FUNCTION_BLOCK Explicit_Controller_FCN_BLK
VAR_INPUT
    ssMethodType: SINT;
    MeasuredTankOutputs: ARRAY [0..1] OF LREAL;
    ref: ARRAY [0..1] OF LREAL;
END_VAR

VAR_OUTPUT
    mv: ARRAY [0..1] OF LREAL;
END_VAR

VAR
    last_x_PreviousInput: ARRAY [0..5] OF LREAL;
    last_mv_DSTATE: ARRAY [0..1] OF LREAL;
    Explicit_b_M: ARRAY [0..11] OF LREAL := [0.00012829320734723115,1.0284618689926092E-5,2.4378658054917943E-5,
        9.19840748563352E-5,0.095123941749644919,1.2151957187730602E-6,2.8085799988137366E-5,0.00013352110274451323,
        9.1481345508264347E-5,2.6760937667881709E-5,-1.5083632311296561E-6,0.095123901802077374];
    Explicit_b_Cm: ARRAY [0..11] OF LREAL := [0.15299877600979192,0.0,0.0,0.15299877600979192,0.0,0.0,0.0,0.0,1.0,
        0.0,0.0,1.0];
    Explicit_b_thmin: ARRAY [0..9] OF LREAL := [-10.0,-14.0,-2.608763482112793,-0.757334910684223,-1.0,-1.0,-12.5,
        -17.5,-6.7801207082609904,-11.7277902321632];
    Explicit_b_thmax: ARRAY [0..9] OF LREAL := [20.0,16.0,27.391236517887208,29.242665089315778,1.0,1.0,25.0,20.0,
        17.219879291739009,12.2722097678368];
    b_i1: ARRAY [0..33] OF INT := [1,23,45,67,87,107,128,148,169,191,211,231,251,271,292,310,332,350,369,391,410,431,
        453,472,492,514,535,554,576,596,616,636,657,676];
    b_i2: ARRAY [0..33] OF INT := [22,44,66,86,106,127,147,168,190,210,230,250,270,291,309,331,349,368,390,409,430,
        452,471,491,513,534,553,575,595,615,635,656,675,697];
    Explicit_c_K: ARRAY [0..696] OF LREAL := [2.0611413896907527,1.9955837259660221,0.261375942086798,
        0.36517295006730383,0.154055652781239,0.21525342211788329,20.0,16.0,27.391236517887208,29.242665089315778,
        1.0,1.0,17.219879291739009,12.2722097678368,10.0,14.0,2.608763482112793,0.757334910684223,1.0,1.0,
        6.7801207082609904,11.7277902321632,-2.0611413896907527,10.306132877927066,2.0017312431194147,
        0.3588547626396722,0.208800889557635,20.0,16.0,27.391236517887208,29.242665089315778,1.0,1.0,25.0,
        17.219879291739009,12.2722097678368,10.0,14.0,2.608763482112793,0.757334910684223,1.0,1.0,
        6.7801207082609904,11.7277902321632,-1.9955837259660218,9.9754498249952146,2.0671005215985825,
        0.25507587776500751,0.14778957157873562,20.0,16.0,27.391236517887208,29.242665089315778,1.0,1.0,20.0,
        17.219879291739009,12.2722097678368,10.0,14.0,2.608763482112793,0.757334910684223,1.0,1.0,
        6.7801207082609904,11.7277902321632,-0.2613759420867981,1.9948353088253725,0.36568008759024018,
        0.010244209084743196,0.21578799487811626,20.0,16.0,27.391236517887208,29.242665089315778,1.0,1.0,
        12.2722097678368,10.0,14.0,2.608763482112793,0.757334910684223,1.0,1.0,6.7801207082609904,11.7277902321632,
        -0.36517295006730388,2.0601920598036507,0.26211153239863794,0.15479976076082763,0.014378493331328977,20.0,
        16.0,27.391236517887208,29.242665089315778,1.0,1.0,17.219879291739009,10.0,14.0,2.608763482112793,
        0.757334910684223,1.0,1.0,6.7801207082609904,11.7277902321632,-0.15405565278123903,1.9948283464872751,
        0.77031009910361337,0.3655913731280393,0.21570378618977479,20.0,16.0,27.391236517887208,29.242665089315778,
        1.0,1.0,17.219879291739009,12.2722097678368,10.0,14.0,2.608763482112793,0.757334910684223,1.0,1.0,12.5,
        11.7277902321632,-0.21525342211788326,2.0601821995500464,0.26201367432910744,1.0760008132237195,
        0.154707893627272,20.0,16.0,27.391236517887208,29.242665089315778,1.0,1.0,17.219879291739009,
        12.2722097678368,10.0,14.0,2.608763482112793,0.757334910684223,1.0,1.0,6.7801207082609904,
        -10.306132877927066,2.0028782849354068,0.35771891427389396,0.20764078266896283,20.0,16.0,27.391236517887208,
        29.242665089315778,1.0,1.0,25.0,17.219879291739009,12.2722097678368,10.0,14.0,2.608763482112793,
        0.757334910684223,1.0,1.0,6.7801207082609904,11.7277902321632,-2.0671005215985825,-2.0017312431194143,
        10.31038937822318,9.979316651871887,20.0,16.0,27.391236517887208,29.242665089315778,1.0,1.0,25.0,20.0,
        17.219879291739009,12.2722097678368,10.0,14.0,2.608763482112793,0.757334910684223,1.0,1.0,
        6.7801207082609904,11.7277902321632,-2.0601920598036503,-0.35885476263967225,10.304338652450928,
        0.0078003539108829258,20.0,16.0,27.391236517887208,29.242665089315778,1.0,1.0,25.0,17.219879291739009,10.0,
        14.0,2.608763482112793,0.757334910684223,1.0,1.0,6.7801207082609904,11.7277902321632,-2.0601821995500464,
        -0.20880088955763496,10.303879948828987,1.0708395480624722,20.0,16.0,27.391236517887208,29.242665089315778,
        1.0,1.0,25.0,17.219879291739009,12.2722097678368,10.0,14.0,2.608763482112793,0.757334910684223,1.0,1.0,
        6.7801207082609904,-9.9754498249952128,2.0680301798015472,0.2541304598084248,0.14685003364909435,20.0,16.0,
        27.391236517887208,29.242665089315778,1.0,1.0,20.0,17.219879291739009,12.2722097678368,10.0,14.0,
        2.608763482112793,0.757334910684223,1.0,1.0,6.7801207082609904,-1.9948353088253725,-0.25507587776500751,
        9.97419631577785,0.0040719490329664855,20.0,16.0,27.391236517887208,29.242665089315778,1.0,1.0,20.0,
        12.2722097678368,10.0,14.0,2.608763482112793,0.757334910684223,1.0,1.0,6.7801207082609904,11.7277902321632,
        -1.9948283464872749,-0.14778957157873562,9.9739050689365616,0.76431342623101861,20.0,16.0,
        27.391236517887208,29.242665089315778,1.0,1.0,20.0,17.219879291739009,12.2722097678368,10.0,14.0,
        2.608763482112793,0.757334910684223,1.0,1.0,12.5,11.7277902321632,-0.26211153239863794,-0.36568008759024018,
        0.010993612348099634,0.014947273027453219,20.0,16.0,27.391236517887208,29.242665089315778,1.0,1.0,10.0,14.0,
        2.608763482112793,0.757334910684223,1.0,1.0,6.7801207082609904,11.7277902321632,-0.77031009910361337,
        -0.010244209084743246,1.9947299388091386,0.36567397657122985,0.21578912879523102,20.0,16.0,
        27.391236517887208,29.242665089315778,1.0,1.0,17.219879291739009,12.2722097678368,10.0,14.0,
        2.608763482112793,0.757334910684223,1.0,1.0,12.5,6.7801207082609904,11.7277902321632,-0.26201367432910749,
        -0.21578799487811628,1.0763493615403084,0.010910348192849671,20.0,16.0,27.391236517887208,
        29.242665089315778,1.0,1.0,12.2722097678368,10.0,14.0,2.608763482112793,0.757334910684223,1.0,1.0,
        6.7801207082609904,-0.36559137312803935,-0.15479976076082763,0.77094478261624777,0.014870549898796829,20.0,
        16.0,27.391236517887208,29.242665089315778,1.0,1.0,17.219879291739009,10.0,14.0,2.608763482112793,
        0.757334910684223,1.0,1.0,12.5,11.7277902321632,-1.0760008132237191,-0.014378493331329066,
        2.0600717378634013,0.26211431296869919,0.15480847558724034,20.0,16.0,27.391236517887208,29.242665089315778,
        1.0,1.0,17.219879291739009,12.2722097678368,10.0,14.0,2.608763482112793,0.757334910684223,1.0,1.0,17.5,
        6.7801207082609904,11.7277902321632,-0.15470789362727197,-0.21570378618977476,0.77082285562521369,
        1.0762511309977898,20.0,16.0,27.391236517887208,29.242665089315778,1.0,1.0,17.219879291739009,
        12.2722097678368,10.0,14.0,2.608763482112793,0.757334910684223,1.0,1.0,12.5,-10.310389378223183,
        -2.0028782849354063,9.9801931781643685,20.0,16.0,27.391236517887208,29.242665089315778,1.0,1.0,25.0,20.0,
        17.219879291739009,12.2722097678368,10.0,14.0,2.608763482112793,0.757334910684223,1.0,1.0,
        6.7801207082609904,11.7277902321632,-10.30433865245093,-0.35771891427389391,-10.303732722383751,
        -1.0699095023920164,20.0,16.0,27.391236517887208,29.242665089315778,1.0,1.0,25.0,17.219879291739009,
        12.2722097678368,10.0,14.0,2.608763482112793,0.757334910684223,1.0,1.0,17.5,6.7801207082609904,
        11.7277902321632,-10.303879948828989,-0.20764078266896283,1.0699095023920167,20.0,16.0,27.391236517887208,
        29.242665089315778,1.0,1.0,25.0,17.219879291739009,12.2722097678368,10.0,14.0,2.608763482112793,
        0.757334910684223,1.0,1.0,6.7801207082609904,-9.9793166518718817,-2.0680301798015472,10.311238407241403,
        20.0,16.0,27.391236517887208,29.242665089315778,1.0,1.0,25.0,20.0,17.219879291739009,12.2722097678368,10.0,
        14.0,2.608763482112793,0.757334910684223,1.0,1.0,6.7801207082609904,-2.0600717378634008,-1.0708395480624708,
        -0.0078003539108829232,10.303732722383758,20.0,16.0,27.391236517887208,29.242665089315778,1.0,1.0,25.0,
        17.219879291739009,12.2722097678368,10.0,14.0,2.608763482112793,0.757334910684223,1.0,1.0,17.5,
        6.7801207082609904,11.7277902321632,-9.9741963157778457,-0.2541304598084248,-9.973787635532247,
        -0.76341041484819772,20.0,16.0,27.391236517887208,29.242665089315778,1.0,1.0,20.0,17.219879291739009,
        12.2722097678368,10.0,14.0,2.608763482112793,0.757334910684223,1.0,1.0,12.5,6.7801207082609904,
        -9.9739050689365616,-0.14685003364909435,0.76341041484819783,20.0,16.0,27.391236517887208,
        29.242665089315778,1.0,1.0,20.0,17.219879291739009,12.2722097678368,10.0,14.0,2.608763482112793,
        0.757334910684223,1.0,1.0,12.5,-1.9947299388091386,-0.76431342623101917,-0.0040719490329664846,
        9.9737876355322488,20.0,16.0,27.391236517887208,29.242665089315778,1.0,1.0,20.0,17.219879291739009,
        12.2722097678368,10.0,14.0,2.608763482112793,0.757334910684223,1.0,1.0,12.5,6.7801207082609904,
        11.7277902321632,-0.77094478261624833,-0.36567397657122985,-0.010993612348099681,0.014958980263312462,20.0,
        16.0,27.391236517887208,29.242665089315778,1.0,1.0,17.219879291739009,10.0,14.0,2.608763482112793,
        0.757334910684223,1.0,1.0,12.5,6.7801207082609904,11.7277902321632,-0.26211431296869925,-1.0763493615403084,
        -0.01494727302745312,0.011010054217011499,20.0,16.0,27.391236517887208,29.242665089315778,1.0,1.0,
        12.2722097678368,10.0,14.0,2.608763482112793,0.757334910684223,1.0,1.0,17.5,6.7801207082609904,
        11.7277902321632,-0.77082285562521369,-0.010910348192849697,-0.215789128795231,1.0763150450241359,20.0,16.0,
        27.391236517887208,29.242665089315778,1.0,1.0,17.219879291739009,12.2722097678368,10.0,14.0,
        2.608763482112793,0.757334910684223,1.0,1.0,12.5,6.7801207082609904,-1.0762511309977894,
        -0.15480847558724031,-0.014870549898796815,0.77091609970584685,20.0,16.0,27.391236517887208,
        29.242665089315778,1.0,1.0,17.219879291739009,12.2722097678368,10.0,14.0,2.608763482112793,
        0.757334910684223,1.0,1.0,12.5,17.5,11.7277902321632,-10.31123840724141,-9.98019317816437,20.0,16.0,
        27.391236517887208,29.242665089315778,1.0,1.0,25.0,20.0,17.219879291739009,12.2722097678368,10.0,14.0,
        2.608763482112793,0.757334910684223,1.0,1.0,6.7801207082609904,-0.77091609970584707,-1.0763150450241361,
        -0.011010054217011499,-0.014958980263312384,20.0,16.0,27.391236517887208,29.242665089315778,1.0,1.0,
        17.219879291739009,12.2722097678368,10.0,14.0,2.608763482112793,0.757334910684223,1.0,1.0,12.5,17.5,
        6.7801207082609904,11.7277902321632];
    Explicit_g_H: ARRAY [0..6969] OF LREAL := [-0.10330544107194929,-0.0014745226031521231,0.10246575755178296,
        0.0015946624161439463,0.10330544107194929,0.0014745226031521231,1.0,0.0,0.0,0.0,0.0,0.0,0.0,0.0,-1.0,-0.0,
        -0.0,-0.0,-0.0,-0.0,-0.0,-0.0,0.10330544107194932,-0.090583151736267742,-0.0017962349061867956,
        0.0019086047501879714,0.0017962349061867956,1.0,0.0,0.0,0.0,0.0,0.0,0.0,0.0,0.0,-1.0,-0.0,-0.0,-0.0,-0.0,
        -0.0,-0.0,-0.0,0.0014745226031521231,-0.0020664403881641815,-0.10329574071922931,0.10245558523686728,
        0.10329574071922931,1.0,0.0,0.0,0.0,0.0,0.0,0.0,0.0,0.0,-1.0,-0.0,-0.0,-0.0,-0.0,-0.0,-0.0,-0.0,
        -0.10246575755178298,-0.0016921077114560436,0.0018070761592905537,0.1036139903469729,0.0016921077114560436,
        1.0,0.0,0.0,0.0,0.0,0.0,0.0,-1.0,-0.0,-0.0,-0.0,-0.0,-0.0,-0.0,-0.0,-0.0015946624161439465,
        -0.10329918232016434,0.10245919014615755,0.10329918232016434,0.0013034270519242509,1.0,0.0,0.0,0.0,0.0,0.0,
        0.0,-1.0,-0.0,-0.0,-0.0,-0.0,-0.0,-0.0,-0.0,-0.10330544107194932,-0.0017962349061867956,
        0.090583151736267742,0.0019086047501879714,0.0017962349061867956,1.0,0.0,0.0,0.0,0.0,0.0,0.0,0.0,-1.0,-0.0,
        -0.0,-0.0,-0.0,-0.0,-0.0,-0.0,-0.0014745226031521231,-0.10329574071922931,0.10245558523686728,
        0.0020664403881641815,0.10329574071922931,1.0,0.0,0.0,0.0,0.0,0.0,0.0,0.0,-1.0,-0.0,-0.0,-0.0,-0.0,-0.0,
        -0.0,0.090583151736267686,-0.0018064099095009775,0.00191855841785106,0.0018064099095009775,1.0,0.0,0.0,0.0,
        0.0,0.0,0.0,0.0,0.0,-1.0,-0.0,-0.0,-0.0,-0.0,-0.0,-0.0,-0.0,0.10329574071922928,0.0017962349061867954,
        -0.090574043803180182,-0.0023185749657277268,1.0,0.0,0.0,0.0,0.0,0.0,0.0,0.0,0.0,0.0,-1.0,-0.0,-0.0,-0.0,
        -0.0,-0.0,-0.0,-0.0,0.10329918232016433,-0.0019086047501879714,-0.090577300277252346,0.0016329685799659197,
        1.0,0.0,0.0,0.0,0.0,0.0,0.0,0.0,-1.0,-0.0,-0.0,-0.0,-0.0,-0.0,-0.0,-0.0,0.10329574071922928,
        -0.0017962349061867954,-0.090574043803180182,0.0023185749657277268,1.0,0.0,0.0,0.0,0.0,0.0,0.0,0.0,0.0,-1.0,
        -0.0,-0.0,-0.0,-0.0,-0.0,-0.0,0.0020664403881641823,-0.10329547444997711,0.1024553070868839,
        0.10329547444997711,1.0,0.0,0.0,0.0,0.0,0.0,0.0,0.0,0.0,-1.0,-0.0,-0.0,-0.0,-0.0,-0.0,-0.0,
        0.0016921077114560436,-0.10245558523686726,-0.0022374573065447505,0.10360521588894454,1.0,0.0,0.0,0.0,0.0,
        0.0,0.0,0.0,-1.0,-0.0,-0.0,-0.0,-0.0,-0.0,-0.0,-0.0,0.0017962349061867956,-0.10329574071922931,
        -0.0023185749657277242,0.090574043803180029,1.0,0.0,0.0,0.0,0.0,0.0,0.0,0.0,0.0,-1.0,-0.0,-0.0,-0.0,-0.0,
        -0.0,-0.0,-0.0,-0.10245919014615754,-0.0018070761592905537,0.10360833927584194,0.0015261960444034593,1.0,
        0.0,0.0,0.0,0.0,0.0,-1.0,-0.0,-0.0,-0.0,-0.0,-0.0,-0.0,-0.0,-0.090583151736267686,-0.1036139903469729,
        -0.0018064099095009775,0.00191855841785106,0.0018064099095009775,1.0,0.0,0.0,0.0,0.0,0.0,0.0,0.0,-1.0,-0.0,
        -0.0,-0.0,-0.0,-0.0,-0.0,-0.0,-0.0,-0.10245558523686728,-0.0016921077114560434,0.0022374573065447496,
        0.10360521588894449,1.0,0.0,0.0,0.0,0.0,0.0,0.0,-1.0,-0.0,-0.0,-0.0,-0.0,-0.0,-0.0,-0.0019086047501879716,
        -0.10329918232016436,0.0905773002772523,0.0016329685799659197,1.0,0.0,0.0,0.0,0.0,0.0,0.0,-1.0,-0.0,-0.0,
        -0.0,-0.0,-0.0,-0.0,-0.0,-0.0020664403881641823,-0.0013034270519242512,-0.10329547444997711,
        0.1024553070868839,0.10329547444997711,1.0,0.0,0.0,0.0,0.0,0.0,0.0,0.0,-1.0,-0.0,-0.0,-0.0,-0.0,-0.0,-0.0,
        -0.0,-0.0,-0.10329574071922928,-0.0017962349061867954,0.090574043803180182,0.0023185749657277268,1.0,0.0,
        0.0,0.0,0.0,0.0,0.0,0.0,-1.0,-0.0,-0.0,-0.0,-0.0,-0.0,-0.0,0.090574043803180043,0.0018064099095009773,
        -0.0023266928925573028,1.0,0.0,0.0,0.0,0.0,0.0,0.0,0.0,0.0,0.0,-1.0,-0.0,-0.0,-0.0,-0.0,-0.0,-0.0,-0.0,
        0.090577300277252346,-0.0019185584178510596,0.090573807363914446,-0.0023266928925573006,1.0,0.0,0.0,0.0,0.0,
        0.0,0.0,0.0,0.0,-1.0,-0.0,-0.0,-0.0,-0.0,-0.0,-0.0,-0.0,-0.0,0.090574043803180043,-0.0018064099095009773,
        0.0023266928925573028,1.0,0.0,0.0,0.0,0.0,0.0,0.0,0.0,0.0,-1.0,-0.0,-0.0,-0.0,-0.0,-0.0,-0.0,
        0.0023185749657277264,0.10329547444997711,-0.09057380736391446,1.0,0.0,0.0,0.0,0.0,0.0,0.0,0.0,0.0,0.0,-1.0,
        -0.0,-0.0,-0.0,-0.0,-0.0,-0.0,0.1032954744499771,-0.0023185749657277247,-0.0016329685799659197,
        -0.0905738073639145,1.0,0.0,0.0,0.0,0.0,0.0,0.0,0.0,0.0,-1.0,-0.0,-0.0,-0.0,-0.0,-0.0,-0.0,-0.0,-0.0,
        0.0022374573065447509,-0.1024553070868839,0.0023266928925573015,-0.090573807363914488,1.0,0.0,0.0,0.0,0.0,
        0.0,0.0,0.0,0.0,-1.0,-0.0,-0.0,-0.0,-0.0,-0.0,-0.0,-0.0,0.0023185749657277255,-0.1032954744499771,
        0.0905738073639145,1.0,0.0,0.0,0.0,0.0,0.0,0.0,0.0,0.0,-1.0,-0.0,-0.0,-0.0,-0.0,-0.0,-0.0,
        0.0018064099095009777,-0.090574043803180057,-0.10360521588894456,-0.0023266928925573011,1.0,0.0,0.0,0.0,0.0,
        0.0,0.0,0.0,0.0,-1.0,-0.0,-0.0,-0.0,-0.0,-0.0,-0.0,-0.0,-0.0,-0.090577300277252318,-0.0019185584178510599,
        -0.10360833927584194,0.0016433588476607495,1.0,0.0,0.0,0.0,0.0,0.0,0.0,-1.0,-0.0,-0.0,-0.0,-0.0,-0.0,-0.0,
        -0.0,-0.0,-0.10245530708688391,-0.0022374573065447492,-0.0015261960444034593,0.10360497454409653,1.0,0.0,
        0.0,0.0,0.0,0.0,0.0,-1.0,-0.0,-0.0,-0.0,-0.0,-0.0,-0.0,-0.0,-0.0,-0.090574043803180043,-0.10360521588894456,
        -0.0018064099095009773,0.0023266928925573028,1.0,0.0,0.0,0.0,0.0,0.0,0.0,0.0,-1.0,-0.0,-0.0,-0.0,-0.0,-0.0,
        -0.0,-0.0,-0.0023185749657277264,-0.10329547444997711,-0.0016329685799659191,0.09057380736391446,1.0,0.0,
        0.0,0.0,0.0,0.0,0.0,0.0,-1.0,-0.0,-0.0,-0.0,-0.0,-0.0,-0.0,-0.0,-0.0,0.090573807363914446,
        0.0023266928925572993,1.0,0.0,0.0,0.0,0.0,0.0,0.0,0.0,0.0,0.0,-1.0,-0.0,-0.0,-0.0,-0.0,-0.0,-0.0,
        -0.090573807363914446,-0.0023266928925572993,-0.10360497454409655,-0.0016433588476607497,1.0,0.0,0.0,0.0,
        0.0,0.0,0.0,0.0,-1.0,-0.0,-0.0,-0.0,-0.0,-0.0,-0.0,-0.0,-0.0,-0.0,-0.0029866651271786876,
        -0.10390116291611282,0.0031875003616156274,0.10304688647343455,0.0029866651271786876,0.10390116291611282,
        0.0,1.0,0.0,0.0,0.0,0.0,0.0,0.0,-0.0,-1.0,-0.0,-0.0,-0.0,-0.0,-0.0,-0.0,0.002986665127178688,
        -0.0039359133245656739,-0.10389613523146926,0.1030418390266099,0.10389613523146926,0.0,1.0,0.0,0.0,0.0,0.0,
        0.0,0.0,0.0,-0.0,-1.0,-0.0,-0.0,-0.0,-0.0,-0.0,-0.0,0.10390116291611282,-0.091095658056062873,
        -0.0033113868084985666,0.0035130907390366621,0.0033113868084985666,0.0,1.0,0.0,0.0,0.0,0.0,0.0,0.0,0.0,-0.0,
        -1.0,-0.0,-0.0,-0.0,-0.0,-0.0,-0.0,-0.0031875003616156279,-0.1038978860866369,0.10304359668322663,
        0.0026964566969657241,0.1038978860866369,0.0,1.0,0.0,0.0,0.0,0.0,0.0,-0.0,-1.0,-0.0,-0.0,-0.0,-0.0,-0.0,
        -0.0,-0.10304688647343456,-0.0032003930853852416,0.0034018852466296103,0.0032003930853852416,
        0.10422852726420227,0.0,1.0,0.0,0.0,0.0,0.0,0.0,-0.0,-1.0,-0.0,-0.0,-0.0,-0.0,-0.0,-0.0,
        -0.002986665127178688,-0.10389613523146926,0.0039359133245656739,0.1030418390266099,0.10389613523146926,0.0,
        1.0,0.0,0.0,0.0,0.0,0.0,0.0,-0.0,-1.0,-0.0,-0.0,-0.0,-0.0,-0.0,-0.0,-0.10390116291611282,
        -0.0033113868084985666,0.0035130907390366621,0.091095658056062873,0.0033113868084985666,0.0,1.0,0.0,0.0,0.0,
        0.0,0.0,0.0,-0.0,-1.0,-0.0,-0.0,-0.0,-0.0,-0.0,0.0039359133245656722,-0.10389596374005793,
        0.10304166986211653,0.10389596374005793,0.0,1.0,0.0,0.0,0.0,0.0,0.0,0.0,0.0,-0.0,-1.0,-0.0,-0.0,-0.0,-0.0,
        -0.0,-0.0,0.0033113868084985666,0.10389613523146926,-0.0042412342413153167,-0.091092939463560868,0.0,1.0,
        0.0,0.0,0.0,0.0,0.0,0.0,0.0,0.0,-0.0,-1.0,-0.0,-0.0,-0.0,-0.0,-0.0,-0.0,0.0032003930853852407,
        -0.10304183902660989,-0.0041373691182175487,0.10422380845249599,0.0,1.0,0.0,0.0,0.0,0.0,0.0,0.0,-0.0,-1.0,
        -0.0,-0.0,-0.0,-0.0,-0.0,-0.0,0.0033113868084985666,-0.10389613523146926,-0.0042412342413153167,
        0.091092939463560868,0.0,1.0,0.0,0.0,0.0,0.0,0.0,0.0,0.0,-0.0,-1.0,-0.0,-0.0,-0.0,-0.0,-0.0,
        0.091095658056062873,-0.0033199458639416968,0.0035216972663637824,0.0033199458639416968,0.0,1.0,0.0,0.0,0.0,
        0.0,0.0,0.0,0.0,-0.0,-1.0,-0.0,-0.0,-0.0,-0.0,-0.0,0.10389788608663691,-0.0035130907390366617,
        -0.0910939728911974,0.0030174925306511403,0.0,1.0,0.0,0.0,0.0,0.0,0.0,0.0,-0.0,-1.0,-0.0,-0.0,-0.0,-0.0,
        -0.0,-0.0,0.10389613523146925,-0.0033113868084985666,-0.091092939463560924,0.0042412342413153123,0.0,1.0,
        0.0,0.0,0.0,0.0,0.0,0.0,0.0,-0.0,-1.0,-0.0,-0.0,-0.0,-0.0,-0.0,-0.0,-0.0034018852466296103,
        -0.10304359668322662,0.0029076453649676762,0.10422546298600668,0.0,1.0,0.0,0.0,0.0,0.0,-0.0,-1.0,-0.0,-0.0,
        -0.0,-0.0,-0.0,-0.0,-0.0039359133245656722,-0.0026964566969657237,-0.10389596374005793,0.10304166986211653,
        0.10389596374005793,0.0,1.0,0.0,0.0,0.0,0.0,0.0,0.0,-0.0,-1.0,-0.0,-0.0,-0.0,-0.0,-0.0,-0.0,-0.0,
        -0.0035130907390366621,-0.1038978860866369,0.091093972891197583,0.0030174925306511377,0.0,1.0,0.0,0.0,0.0,
        0.0,0.0,-0.0,-1.0,-0.0,-0.0,-0.0,-0.0,-0.0,-0.1030418390266099,-0.0032003930853852416,0.0041373691182175461,
        0.10422380845249597,0.0,1.0,0.0,0.0,0.0,0.0,0.0,-0.0,-1.0,-0.0,-0.0,-0.0,-0.0,-0.0,-0.0,
        -0.091095658056062873,-0.10422852726420226,-0.0033199458639416968,0.0035216972663637824,
        0.0033199458639416968,0.0,1.0,0.0,0.0,0.0,0.0,0.0,0.0,-0.0,-1.0,-0.0,-0.0,-0.0,-0.0,-0.0,-0.0,-0.0,
        -0.0033113868084985666,-0.10389613523146926,0.0042412342413153167,0.091092939463560868,0.0,1.0,0.0,0.0,0.0,
        0.0,0.0,0.0,-0.0,-1.0,-0.0,-0.0,-0.0,-0.0,-0.0,0.0042412342413153149,0.10389596374005791,
        -0.09109287411848567,0.0,1.0,0.0,0.0,0.0,0.0,0.0,0.0,0.0,0.0,-0.0,-1.0,-0.0,-0.0,-0.0,-0.0,-0.0,-0.0,
        0.0041373691182175452,-0.10304166986211651,0.0042494263649640318,-0.0910928741184855,0.0,1.0,0.0,0.0,0.0,
        0.0,0.0,0.0,0.0,-0.0,-1.0,-0.0,-0.0,-0.0,-0.0,-0.0,-0.0,-0.0,0.0042412342413153149,-0.10389596374005791,
        0.09109287411848567,0.0,1.0,0.0,0.0,0.0,0.0,0.0,0.0,0.0,-0.0,-1.0,-0.0,-0.0,-0.0,-0.0,-0.0,
        0.0910929394635609,0.0033199458639416963,-0.0042494263649640335,0.0,1.0,0.0,0.0,0.0,0.0,0.0,0.0,0.0,0.0,
        -0.0,-1.0,-0.0,-0.0,-0.0,-0.0,-0.0,0.0033199458639416959,-0.091092939463561,-0.10422380845249592,
        -0.004249426364964037,0.0,1.0,0.0,0.0,0.0,0.0,0.0,0.0,0.0,-0.0,-1.0,-0.0,-0.0,-0.0,-0.0,-0.0,-0.0,-0.0,
        0.0910939728911976,-0.0035216972663637829,0.091092874118485587,-0.0042494263649640309,0.0,1.0,0.0,0.0,0.0,
        0.0,0.0,0.0,0.0,-0.0,-1.0,-0.0,-0.0,-0.0,-0.0,-0.0,-0.0,0.0910929394635609,-0.0033199458639416968,
        0.0042494263649640318,0.0,1.0,0.0,0.0,0.0,0.0,0.0,0.0,0.0,-0.0,-1.0,-0.0,-0.0,-0.0,-0.0,-0.0,
        0.10389596374005794,-0.0042412342413153132,-0.0030174925306511394,-0.091092874118485587,0.0,1.0,0.0,0.0,0.0,
        0.0,0.0,0.0,0.0,-0.0,-1.0,-0.0,-0.0,-0.0,-0.0,-0.0,-0.0,-0.0,-0.0041373691182175444,-0.10304166986211653,
        -0.0029076453649676775,0.10422364519688854,0.0,1.0,0.0,0.0,0.0,0.0,0.0,-0.0,-1.0,-0.0,-0.0,-0.0,-0.0,-0.0,
        -0.0,-0.0,-0.0035216972663637833,-0.091093972891197486,-0.10422546298600667,0.00302592181600906,0.0,1.0,0.0,
        0.0,0.0,0.0,0.0,-0.0,-1.0,-0.0,-0.0,-0.0,-0.0,-0.0,-0.0,-0.0,-0.0042412342413153149,-0.0030174925306511386,
        -0.10389596374005791,0.09109287411848567,0.0,1.0,0.0,0.0,0.0,0.0,0.0,0.0,-0.0,-1.0,-0.0,-0.0,-0.0,-0.0,-0.0,
        -0.0,-0.0910929394635609,-0.0033199458639416963,-0.10422380845249594,0.0042494263649640335,0.0,1.0,0.0,0.0,
        0.0,0.0,0.0,0.0,-0.0,-1.0,-0.0,-0.0,-0.0,-0.0,-0.0,-0.0,-0.0,0.0042494263649640335,0.091092874118485545,0.0,
        1.0,0.0,0.0,0.0,0.0,0.0,0.0,0.0,0.0,-0.0,-1.0,-0.0,-0.0,-0.0,-0.0,-0.0,-0.0042494263649640335,
        -0.091092874118485545,-0.00302592181600906,-0.10422364519688854,0.0,1.0,0.0,0.0,0.0,0.0,0.0,0.0,-0.0,-1.0,
        -0.0,-0.0,-0.0,-0.0,-0.0,-0.0,-0.0,-0.0,-0.0071014157036083953,-0.00011441872526747157,
        0.0068071732563204012,0.00012053113664926074,0.0071014157036083953,0.00011441872526747157,0.0,0.0,1.0,0.0,
        0.0,0.0,0.0,0.0,-0.0,-0.0,-1.0,-0.0,-0.0,-0.0,-0.0,-0.0,0.0071014157036083962,-0.0048430438770123655,
        -0.00013653204941286985,0.00014211064337640565,0.00013653204941286985,0.0,0.0,1.0,0.0,0.0,0.0,0.0,0.0,0.0,
        -0.0,-0.0,-1.0,-0.0,-0.0,-0.0,-0.0,-0.0,0.00011441872526747157,-0.000141573042344912,-0.0071007897421819293,
        0.0068065491278817619,0.0071007897421819293,0.0,0.0,1.0,0.0,0.0,0.0,0.0,0.0,0.0,-0.0,-0.0,-1.0,-0.0,-0.0,
        -0.0,-0.0,-0.0,-0.0068071732563204021,-0.00012887210385476621,0.00013464115259381751,0.0074369160608808611,
        0.00012887210385476621,0.0,0.0,1.0,0.0,0.0,0.0,0.0,-0.0,-0.0,-1.0,-0.0,-0.0,-0.0,-0.0,-0.0,
        -0.00012053113664926074,-0.0071010081244634151,0.00680676736109825,0.0071010081244634151,
        0.00010540752661209963,0.0,0.0,1.0,0.0,0.0,0.0,0.0,-0.0,-0.0,-1.0,-0.0,-0.0,-0.0,-0.0,-0.0,
        -0.0071014157036083962,-0.00013653204941286985,0.0048430438770123655,0.00014211064337640565,
        0.00013653204941286985,0.0,0.0,1.0,0.0,0.0,0.0,0.0,0.0,-0.0,-0.0,-1.0,-0.0,-0.0,-0.0,-0.0,-0.0,
        -0.00011441872526747157,-0.0071007897421819293,0.0068065491278817619,0.000141573042344912,
        0.0071007897421819293,0.0,0.0,1.0,0.0,0.0,0.0,0.0,0.0,-0.0,-0.0,-1.0,-0.0,-0.0,-0.0,-0.0,
        0.004843043877012362,-0.0001370758183784174,0.00014264258380223117,0.0001370758183784174,0.0,0.0,1.0,0.0,
        0.0,0.0,0.0,0.0,0.0,-0.0,-0.0,-1.0,-0.0,-0.0,-0.0,-0.0,-0.0,0.0071007897421819293,0.00013653204941286982,
        -0.00484267616986334,-0.00015890541712753912,0.0,0.0,1.0,0.0,0.0,0.0,0.0,0.0,0.0,0.0,-0.0,-0.0,-1.0,-0.0,
        -0.0,-0.0,-0.0,-0.0,0.0071010081244634142,-0.00014211064337640562,-0.0048428095237973432,
        0.00012805865559832721,0.0,0.0,1.0,0.0,0.0,0.0,0.0,0.0,-0.0,-0.0,-1.0,-0.0,-0.0,-0.0,-0.0,-0.0,
        0.0071007897421819293,-0.00013653204941286982,-0.00484267616986334,0.00015890541712753912,0.0,0.0,1.0,0.0,
        0.0,0.0,0.0,0.0,0.0,-0.0,-0.0,-1.0,-0.0,-0.0,-0.0,-0.0,0.00014157304234491195,-0.0071007713931416907,
        0.0068065310553807263,0.0071007713931416907,0.0,0.0,1.0,0.0,0.0,0.0,0.0,0.0,0.0,-0.0,-0.0,-1.0,-0.0,-0.0,
        -0.0,-0.0,0.00012887210385476621,-0.006806549127881761,-0.00015293404910673837,0.0074363092277326959,0.0,
        0.0,1.0,0.0,0.0,0.0,0.0,0.0,-0.0,-0.0,-1.0,-0.0,-0.0,-0.0,-0.0,-0.0,0.00013653204941286982,
        -0.00710078974218193,-0.00015890541712753893,0.0048426761698633393,0.0,0.0,1.0,0.0,0.0,0.0,0.0,0.0,0.0,-0.0,
        -0.0,-1.0,-0.0,-0.0,-0.0,-0.0,-0.0,-0.0068067673610982512,-0.00013464115259381751,0.0074365205859498427,
        0.0001202050585799296,0.0,0.0,1.0,0.0,0.0,0.0,-0.0,-0.0,-1.0,-0.0,-0.0,-0.0,-0.0,-0.0,-0.004843043877012362,
        -0.0074369160608808611,-0.0001370758183784174,0.00014264258380223117,0.0001370758183784174,0.0,0.0,1.0,0.0,
        0.0,0.0,0.0,0.0,-0.0,-0.0,-1.0,-0.0,-0.0,-0.0,-0.0,-0.0,-0.0,-0.0068065491278817619,-0.00012887210385476621,
        0.00015293404910673842,0.0074363092277326941,0.0,0.0,1.0,0.0,0.0,0.0,0.0,-0.0,-0.0,-1.0,-0.0,-0.0,-0.0,-0.0,
        -0.00014211064337640565,-0.0071010081244634159,0.0048428095237973406,0.00012805865559832721,0.0,0.0,1.0,0.0,
        0.0,0.0,0.0,-0.0,-0.0,-1.0,-0.0,-0.0,-0.0,-0.0,-0.0,-0.00014157304234491195,-0.00010540752661209965,
        -0.0071007713931416907,0.0068065310553807263,0.0071007713931416907,0.0,0.0,1.0,0.0,0.0,0.0,0.0,0.0,-0.0,
        -0.0,-1.0,-0.0,-0.0,-0.0,-0.0,-0.0,-0.0,-0.0071007897421819293,-0.00013653204941286982,0.00484267616986334,
        0.00015890541712753912,0.0,0.0,1.0,0.0,0.0,0.0,0.0,0.0,-0.0,-0.0,-1.0,-0.0,-0.0,-0.0,-0.0,
        0.0048426761698633488,0.0001370758183784174,-0.00015933928310827815,0.0,0.0,1.0,0.0,0.0,0.0,0.0,0.0,0.0,0.0,
        -0.0,-0.0,-1.0,-0.0,-0.0,-0.0,-0.0,-0.0,0.0048428095237973475,-0.00014264258380223112,0.0048426666784349339,
        -0.00015933928310827783,0.0,0.0,1.0,0.0,0.0,0.0,0.0,0.0,0.0,-0.0,-0.0,-1.0,-0.0,-0.0,-0.0,-0.0,-0.0,-0.0,
        0.0048426761698633488,-0.0001370758183784174,0.00015933928310827815,0.0,0.0,1.0,0.0,0.0,0.0,0.0,0.0,0.0,
        -0.0,-0.0,-1.0,-0.0,-0.0,-0.0,-0.0,0.00015890541712753904,0.0071007713931416925,-0.0048426666784349322,0.0,
        0.0,1.0,0.0,0.0,0.0,0.0,0.0,0.0,0.0,-0.0,-0.0,-1.0,-0.0,-0.0,-0.0,-0.0,0.00710077139314169,
        -0.00015890541712753904,-0.00012805865559832719,-0.0048426666784349417,0.0,0.0,1.0,0.0,0.0,0.0,0.0,0.0,0.0,
        -0.0,-0.0,-1.0,-0.0,-0.0,-0.0,-0.0,-0.0,-0.0,0.00015293404910673837,-0.0068065310553807254,
        0.000159339283108278,-0.0048426666784349304,0.0,0.0,1.0,0.0,0.0,0.0,0.0,0.0,0.0,-0.0,-0.0,-1.0,-0.0,-0.0,
        -0.0,-0.0,-0.0,0.000158905417127539,-0.00710077139314169,0.0048426666784349348,0.0,0.0,1.0,0.0,0.0,0.0,0.0,
        0.0,0.0,-0.0,-0.0,-1.0,-0.0,-0.0,-0.0,-0.0,0.0001370758183784174,-0.0048426761698633454,
        -0.0074363092277326967,-0.0001593392831082781,0.0,0.0,1.0,0.0,0.0,0.0,0.0,0.0,0.0,-0.0,-0.0,-1.0,-0.0,-0.0,
        -0.0,-0.0,-0.0,-0.0,-0.0048428095237973458,-0.00014264258380223115,-0.0074365205859498436,
        0.00012861393248801036,0.0,0.0,1.0,0.0,0.0,0.0,0.0,-0.0,-0.0,-1.0,-0.0,-0.0,-0.0,-0.0,-0.0,-0.0,
        -0.0068065310553807271,-0.00015293404910673839,-0.00012020505857992958,0.0074362911951540191,0.0,0.0,1.0,
        0.0,0.0,0.0,0.0,-0.0,-0.0,-1.0,-0.0,-0.0,-0.0,-0.0,-0.0,-0.0,-0.0048426761698633488,-0.007436309227732695,
        -0.0001370758183784174,0.00015933928310827815,0.0,0.0,1.0,0.0,0.0,0.0,0.0,0.0,-0.0,-0.0,-1.0,-0.0,-0.0,-0.0,
        -0.0,-0.0,-0.00015890541712753904,-0.0071007713931416925,-0.00012805865559832716,0.0048426666784349322,0.0,
        0.0,1.0,0.0,0.0,0.0,0.0,0.0,-0.0,-0.0,-1.0,-0.0,-0.0,-0.0,-0.0,-0.0,-0.0,0.004842666678434933,
        0.00015933928310827788,0.0,0.0,1.0,0.0,0.0,0.0,0.0,0.0,0.0,0.0,-0.0,-0.0,-1.0,-0.0,-0.0,-0.0,-0.0,
        -0.004842666678434933,-0.00015933928310827788,-0.00743629119515402,-0.00012861393248801042,0.0,0.0,1.0,0.0,
        0.0,0.0,0.0,0.0,-0.0,-0.0,-1.0,-0.0,-0.0,-0.0,-0.0,-0.0,-0.0,-0.0,-0.00040913205147735833,
        -0.012803913199114694,0.00042684709847512454,0.012280530787446623,0.00040913205147735833,
        0.012803913199114694,0.0,0.0,0.0,1.0,0.0,0.0,0.0,0.0,-0.0,-0.0,-0.0,-1.0,-0.0,-0.0,-0.0,-0.0,
        0.00040913205147735839,-0.00048184876971232865,-0.012803421641857477,0.012280091043666855,
        0.012803421641857477,0.0,0.0,0.0,1.0,0.0,0.0,0.0,0.0,0.0,-0.0,-0.0,-0.0,-1.0,-0.0,-0.0,-0.0,-0.0,
        0.012803913199114692,-0.0087802267724355568,-0.00044914235230113112,0.00046696522506884096,
        0.00044914235230113112,0.0,0.0,0.0,1.0,0.0,0.0,0.0,0.0,0.0,-0.0,-0.0,-0.0,-1.0,-0.0,-0.0,-0.0,-0.0,
        -0.00042684709847512465,-0.012803581733992975,0.012280236188633492,0.00038239527547962392,
        0.012803581733992975,0.0,0.0,0.0,1.0,0.0,0.0,0.0,-0.0,-0.0,-0.0,-1.0,-0.0,-0.0,-0.0,-0.0,
        -0.012280530787446625,-0.00043459798254794492,0.00045239171239116143,0.00043459798254794492,
        0.013399805276596607,0.0,0.0,0.0,1.0,0.0,0.0,0.0,-0.0,-0.0,-0.0,-1.0,-0.0,-0.0,-0.0,-0.0,
        -0.00040913205147735839,-0.012803421641857477,0.00048184876971232865,0.012280091043666855,
        0.012803421641857477,0.0,0.0,0.0,1.0,0.0,0.0,0.0,0.0,-0.0,-0.0,-0.0,-1.0,-0.0,-0.0,-0.0,-0.0,
        -0.012803913199114692,-0.00044914235230113112,0.00046696522506884096,0.0087802267724355568,
        0.00044914235230113112,0.0,0.0,0.0,1.0,0.0,0.0,0.0,0.0,-0.0,-0.0,-0.0,-1.0,-0.0,-0.0,-0.0,
        0.00048184876971232816,-0.012803400150311305,0.012280072289609674,0.012803400150311305,0.0,0.0,0.0,1.0,0.0,
        0.0,0.0,0.0,0.0,-0.0,-0.0,-0.0,-1.0,-0.0,-0.0,-0.0,-0.0,0.00044914235230113112,0.012803421641857476,
        -0.00051947485679715278,-0.0087802823071337216,0.0,0.0,0.0,1.0,0.0,0.0,0.0,0.0,0.0,0.0,-0.0,-0.0,-0.0,-1.0,
        -0.0,-0.0,-0.0,-0.0,0.00043459798254794486,-0.012280091043666853,-0.00050585606663743662,
        0.013399272511122719,0.0,0.0,0.0,1.0,0.0,0.0,0.0,0.0,-0.0,-0.0,-0.0,-1.0,-0.0,-0.0,-0.0,-0.0,
        0.00044914235230113112,-0.012803421641857476,-0.00051947485679715278,0.0087802823071337216,0.0,0.0,0.0,1.0,
        0.0,0.0,0.0,0.0,0.0,-0.0,-0.0,-0.0,-1.0,-0.0,-0.0,-0.0,0.00878022677243555,-0.00044996673444029655,
        0.000467794169019148,0.00044996673444029655,0.0,0.0,0.0,1.0,0.0,0.0,0.0,0.0,0.0,-0.0,-0.0,-0.0,-1.0,-0.0,
        -0.0,-0.0,0.012803581733992975,-0.00046696522506884091,-0.0087802788142219718,0.00042195050475040259,0.0,
        0.0,0.0,1.0,0.0,0.0,0.0,0.0,-0.0,-0.0,-0.0,-1.0,-0.0,-0.0,-0.0,-0.0,0.012803421641857476,
        -0.00044914235230113117,-0.0087802823071337164,0.00051947485679715191,0.0,0.0,0.0,1.0,0.0,0.0,0.0,0.0,0.0,
        -0.0,-0.0,-0.0,-1.0,-0.0,-0.0,-0.0,-0.0,-0.00045239171239116148,-0.012280236188633491,
        0.00040755820299425842,0.013399444045468174,0.0,0.0,0.0,1.0,0.0,0.0,-0.0,-0.0,-0.0,-1.0,-0.0,-0.0,-0.0,-0.0,
        -0.00048184876971232816,-0.000382395275479624,-0.012803400150311305,0.012280072289609674,
        0.012803400150311305,0.0,0.0,0.0,1.0,0.0,0.0,0.0,0.0,-0.0,-0.0,-0.0,-1.0,-0.0,-0.0,-0.0,-0.0,-0.0,
        -0.00046696522506884091,-0.012803581733992975,0.0087802788142219822,0.00042195050475040254,0.0,0.0,0.0,1.0,
        0.0,0.0,0.0,-0.0,-0.0,-0.0,-1.0,-0.0,-0.0,-0.0,-0.012280091043666855,-0.00043459798254794492,
        0.00050585606663743629,0.013399272511122717,0.0,0.0,0.0,1.0,0.0,0.0,0.0,-0.0,-0.0,-0.0,-1.0,-0.0,-0.0,-0.0,
        -0.0,-0.00878022677243555,-0.013399805276596607,-0.00044996673444029655,0.000467794169019148,
        0.00044996673444029655,0.0,0.0,0.0,1.0,0.0,0.0,0.0,0.0,-0.0,-0.0,-0.0,-1.0,-0.0,-0.0,-0.0,-0.0,-0.0,
        -0.00044914235230113112,-0.012803421641857476,0.00051947485679715278,0.0087802823071337216,0.0,0.0,0.0,1.0,
        0.0,0.0,0.0,0.0,-0.0,-0.0,-0.0,-1.0,-0.0,-0.0,-0.0,0.00051947485679715256,0.012803400150311308,
        -0.0087802859415915882,0.0,0.0,0.0,1.0,0.0,0.0,0.0,0.0,0.0,0.0,-0.0,-0.0,-0.0,-1.0,-0.0,-0.0,-0.0,-0.0,
        0.00050585606663743619,-0.012280072289609669,0.00052026393633152477,-0.00878028594159158,0.0,0.0,0.0,1.0,
        0.0,0.0,0.0,0.0,0.0,-0.0,-0.0,-0.0,-1.0,-0.0,-0.0,-0.0,-0.0,-0.0,0.00051947485679715256,
        -0.012803400150311308,0.0087802859415915882,0.0,0.0,0.0,1.0,0.0,0.0,0.0,0.0,0.0,-0.0,-0.0,-0.0,-1.0,-0.0,
        -0.0,-0.0,0.0087802823071337164,0.00044996673444029644,-0.0005202639363315252,0.0,0.0,0.0,1.0,0.0,0.0,0.0,
        0.0,0.0,0.0,-0.0,-0.0,-0.0,-1.0,-0.0,-0.0,-0.0,0.00044996673444029655,-0.0087802823071337112,
        -0.013399272511122719,-0.00052026393633152455,0.0,0.0,0.0,1.0,0.0,0.0,0.0,0.0,0.0,-0.0,-0.0,-0.0,-1.0,-0.0,
        -0.0,-0.0,-0.0,-0.0,0.0087802788142219909,-0.00046779416901914796,0.0087802859415916073,
        -0.00052026393633152531,0.0,0.0,0.0,1.0,0.0,0.0,0.0,0.0,0.0,-0.0,-0.0,-0.0,-1.0,-0.0,-0.0,-0.0,-0.0,
        0.0087802823071337233,-0.0004499667344402965,0.00052026393633152542,0.0,0.0,0.0,1.0,0.0,0.0,0.0,0.0,0.0,
        -0.0,-0.0,-0.0,-1.0,-0.0,-0.0,-0.0,0.012803400150311306,-0.00051947485679715234,-0.0004219505047504027,
        -0.0087802859415915917,0.0,0.0,0.0,1.0,0.0,0.0,0.0,0.0,0.0,-0.0,-0.0,-0.0,-1.0,-0.0,-0.0,-0.0,-0.0,-0.0,
        -0.000505856066637436,-0.012280072289609674,-0.00040755820299425859,0.013399248530954264,0.0,0.0,0.0,1.0,
        0.0,0.0,0.0,-0.0,-0.0,-0.0,-1.0,-0.0,-0.0,-0.0,-0.0,-0.0,-0.000467794169019148,-0.0087802788142219753,
        -0.013399444045468176,0.00042276241085400672,0.0,0.0,0.0,1.0,0.0,0.0,0.0,-0.0,-0.0,-0.0,-1.0,-0.0,-0.0,-0.0,
        -0.0,-0.0,-0.00051947485679715256,-0.00042195050475040254,-0.012803400150311308,0.0087802859415915882,0.0,
        0.0,0.0,1.0,0.0,0.0,0.0,0.0,-0.0,-0.0,-0.0,-1.0,-0.0,-0.0,-0.0,-0.0,-0.0087802823071337164,
        -0.00044996673444029644,-0.013399272511122716,0.0005202639363315252,0.0,0.0,0.0,1.0,0.0,0.0,0.0,0.0,-0.0,
        -0.0,-0.0,-1.0,-0.0,-0.0,-0.0,-0.0,-0.0,0.00052026393633152488,0.0087802859415915847,0.0,0.0,0.0,1.0,0.0,
        0.0,0.0,0.0,0.0,0.0,-0.0,-0.0,-0.0,-1.0,-0.0,-0.0,-0.0,-0.00052026393633152488,-0.0087802859415915847,
        -0.00042276241085400677,-0.013399248530954271,0.0,0.0,0.0,1.0,0.0,0.0,0.0,0.0,-0.0,-0.0,-0.0,-1.0,-0.0,-0.0,
        -0.0,-0.0,-0.0,-0.0,-0.699842938730663,-0.010035599503395155,0.69332035945645,0.010841852728168152,
        0.699842938730663,0.010035599503395155,0.0,0.0,0.0,0.0,1.0,0.0,0.0,0.0,-0.0,-0.0,-0.0,-0.0,-1.0,-0.0,-0.0,
        -0.0,0.69984293873066306,-0.60877543705459958,-0.012215033803492436,0.012968650442024339,
        0.012215033803492436,0.0,0.0,0.0,0.0,1.0,0.0,0.0,0.0,0.0,-0.0,-0.0,-0.0,-0.0,-1.0,-0.0,-0.0,-0.0,
        0.010035599503395155,-0.013997402719325952,-0.69977736900234788,0.6932517133063042,0.69977736900234788,0.0,
        0.0,0.0,0.0,1.0,0.0,0.0,0.0,0.0,-0.0,-0.0,-0.0,-0.0,-1.0,-0.0,-0.0,-0.0,-0.6933203594564501,
        -0.01150785335521526,0.0122791159302254,0.703041617134732,0.01150785335521526,0.0,0.0,0.0,0.0,1.0,0.0,0.0,
        -0.0,-0.0,-0.0,-0.0,-1.0,-0.0,-0.0,-0.0,-0.010841852728168152,-0.69980061939953575,0.69327602991798487,
        0.69980061939953575,0.0088862950073843542,0.0,0.0,0.0,0.0,1.0,0.0,0.0,-0.0,-0.0,-0.0,-0.0,-1.0,-0.0,-0.0,
        -0.0,-0.69984293873066306,-0.012215033803492436,0.60877543705459958,0.012968650442024339,
        0.012215033803492436,0.0,0.0,0.0,0.0,1.0,0.0,0.0,0.0,-0.0,-0.0,-0.0,-0.0,-1.0,-0.0,-0.0,-0.0,
        -0.010035599503395155,-0.69977736900234788,0.6932517133063042,0.013997402719325952,0.69977736900234788,0.0,
        0.0,0.0,0.0,1.0,0.0,0.0,0.0,-0.0,-0.0,-0.0,-0.0,-1.0,-0.0,-0.0,0.60877543705459958,-0.012283415343526595,
        0.0130355444868211,0.012283415343526595,0.0,0.0,0.0,0.0,1.0,0.0,0.0,0.0,0.0,-0.0,-0.0,-0.0,-0.0,-1.0,-0.0,
        -0.0,-0.0,0.69977736900234788,0.012215033803492436,-0.60871464776796336,-0.015705489529037081,0.0,0.0,0.0,
        0.0,1.0,0.0,0.0,0.0,0.0,0.0,-0.0,-0.0,-0.0,-0.0,-1.0,-0.0,-0.0,-0.0,0.69980061939953575,
        -0.012968650442024337,-0.60873638906724648,0.011118767018001796,0.0,0.0,0.0,0.0,1.0,0.0,0.0,0.0,-0.0,-0.0,
        -0.0,-0.0,-1.0,-0.0,-0.0,-0.0,0.69977736900234788,-0.012215033803492436,-0.60871464776796336,
        0.015705489529037081,0.0,0.0,0.0,0.0,1.0,0.0,0.0,0.0,0.0,-0.0,-0.0,-0.0,-0.0,-1.0,-0.0,-0.0,
        0.013997402719325936,-0.699775564999848,0.69324983267331119,0.699775564999848,0.0,0.0,0.0,0.0,1.0,0.0,0.0,
        0.0,0.0,-0.0,-0.0,-0.0,-0.0,-1.0,-0.0,-0.0,0.011507853355215258,-0.69325171330630408,-0.015154564068334616,
        0.70298216286030424,0.0,0.0,0.0,0.0,1.0,0.0,0.0,0.0,-0.0,-0.0,-0.0,-0.0,-1.0,-0.0,-0.0,-0.0,
        0.012215033803492434,-0.69977736900234788,-0.015705489529037078,0.60871464776796369,0.0,0.0,0.0,0.0,1.0,0.0,
        0.0,0.0,0.0,-0.0,-0.0,-0.0,-0.0,-1.0,-0.0,-0.0,-0.0,-0.69327602991798487,-0.0122791159302254,
        0.703003309895513,0.010393624070932634,0.0,0.0,0.0,0.0,1.0,0.0,-0.0,-0.0,-0.0,-0.0,-1.0,-0.0,-0.0,-0.0,
        -0.60877543705459958,-0.703041617134732,-0.012283415343526595,0.0130355444868211,0.012283415343526595,0.0,
        0.0,0.0,0.0,1.0,0.0,0.0,0.0,-0.0,-0.0,-0.0,-0.0,-1.0,-0.0,-0.0,-0.0,-0.0,-0.69325171330630408,
        -0.01150785335521526,0.015154564068334596,0.70298216286030424,0.0,0.0,0.0,0.0,1.0,0.0,0.0,-0.0,-0.0,-0.0,
        -0.0,-1.0,-0.0,-0.0,-0.012968650442024339,-0.69980061939953575,0.60873638906724659,0.011118767018001793,0.0,
        0.0,0.0,0.0,1.0,0.0,0.0,-0.0,-0.0,-0.0,-0.0,-1.0,-0.0,-0.0,-0.0,-0.013997402719325936,
        -0.0088862950073843577,-0.699775564999848,0.69324983267331119,0.699775564999848,0.0,0.0,0.0,0.0,1.0,0.0,0.0,
        0.0,-0.0,-0.0,-0.0,-0.0,-1.0,-0.0,-0.0,-0.0,-0.0,-0.69977736900234788,-0.012215033803492436,
        0.60871464776796336,0.015705489529037081,0.0,0.0,0.0,0.0,1.0,0.0,0.0,0.0,-0.0,-0.0,-0.0,-0.0,-1.0,-0.0,-0.0,
        0.60871464776796325,0.012283415343526595,-0.015760046509446644,0.0,0.0,0.0,0.0,1.0,0.0,0.0,0.0,0.0,0.0,-0.0,
        -0.0,-0.0,-0.0,-1.0,-0.0,-0.0,-0.0,0.60873638906724625,-0.013035544486821099,0.60871306985531193,
        -0.015760046509446641,0.0,0.0,0.0,0.0,1.0,0.0,0.0,0.0,0.0,-0.0,-0.0,-0.0,-0.0,-1.0,-0.0,-0.0,-0.0,-0.0,
        0.60871464776796325,-0.012283415343526595,0.015760046509446644,0.0,0.0,0.0,0.0,1.0,0.0,0.0,0.0,0.0,-0.0,
        -0.0,-0.0,-0.0,-1.0,-0.0,-0.0,0.015705489529037078,0.69977556499984794,-0.60871306985531193,0.0,0.0,0.0,0.0,
        1.0,0.0,0.0,0.0,0.0,0.0,-0.0,-0.0,-0.0,-0.0,-1.0,-0.0,-0.0,0.699775564999848,-0.015705489529037067,
        -0.011118767018001791,-0.60871306985531182,0.0,0.0,0.0,0.0,1.0,0.0,0.0,0.0,0.0,-0.0,-0.0,-0.0,-0.0,-1.0,
        -0.0,-0.0,-0.0,-0.0,0.015154564068334596,-0.69324983267331119,0.015760046509446651,-0.60871306985531182,0.0,
        0.0,0.0,0.0,1.0,0.0,0.0,0.0,0.0,-0.0,-0.0,-0.0,-0.0,-1.0,-0.0,-0.0,-0.0,0.015705489529037074,
        -0.699775564999848,0.60871306985531182,0.0,0.0,0.0,0.0,1.0,0.0,0.0,0.0,0.0,-0.0,-0.0,-0.0,-0.0,-1.0,-0.0,
        -0.0,0.012283415343526595,-0.60871464776796358,-0.70298216286030424,-0.015760046509446644,0.0,0.0,0.0,0.0,
        1.0,0.0,0.0,0.0,0.0,-0.0,-0.0,-0.0,-0.0,-1.0,-0.0,-0.0,-0.0,-0.0,-0.60873638906724625,-0.013035544486821102,
        -0.703003309895513,0.011188595264481212,0.0,0.0,0.0,0.0,1.0,0.0,0.0,-0.0,-0.0,-0.0,-0.0,-1.0,-0.0,-0.0,-0.0,
        -0.0,-0.69324983267331119,-0.015154564068334604,-0.010393624070932634,0.70298052278183043,0.0,0.0,0.0,0.0,
        1.0,0.0,0.0,-0.0,-0.0,-0.0,-0.0,-1.0,-0.0,-0.0,-0.0,-0.0,-0.60871464776796325,-0.70298216286030424,
        -0.012283415343526595,0.015760046509446644,0.0,0.0,0.0,0.0,1.0,0.0,0.0,0.0,-0.0,-0.0,-0.0,-0.0,-1.0,-0.0,
        -0.0,-0.0,-0.015705489529037078,-0.69977556499984794,-0.011118767018001789,0.60871306985531193,0.0,0.0,0.0,
        0.0,1.0,0.0,0.0,0.0,-0.0,-0.0,-0.0,-0.0,-1.0,-0.0,-0.0,-0.0,-0.0,0.60871306985531182,0.015760046509446641,
        0.0,0.0,0.0,0.0,1.0,0.0,0.0,0.0,0.0,0.0,-0.0,-0.0,-0.0,-0.0,-1.0,-0.0,-0.0,-0.60871306985531182,
        -0.015760046509446641,-0.70298052278183043,-0.011188595264481214,0.0,0.0,0.0,0.0,1.0,0.0,0.0,0.0,-0.0,-0.0,
        -0.0,-0.0,-1.0,-0.0,-0.0,-0.0,-0.0,-0.0,-0.020191746911356029,-0.69999450696241372,0.021532772716851709,
        0.6935356133979842,0.020191746911356029,0.69999450696241372,0.0,0.0,0.0,0.0,0.0,1.0,0.0,0.0,-0.0,-0.0,-0.0,
        -0.0,-0.0,-1.0,-0.0,-0.0,0.020191746911356032,-0.026511280680507922,-0.69996085369453254,
        0.69350191818893769,0.69996085369453254,0.0,0.0,0.0,0.0,0.0,1.0,0.0,0.0,0.0,-0.0,-0.0,-0.0,-0.0,-0.0,-1.0,
        -0.0,-0.0,0.69999450696241372,-0.609607128237397,-0.022379425814583805,0.023726305453859561,
        0.022379425814583805,0.0,0.0,0.0,0.0,0.0,1.0,0.0,0.0,0.0,-0.0,-0.0,-0.0,-0.0,-0.0,-1.0,-0.0,-0.0,
        -0.021532772716851712,-0.69997255424705462,0.69351363803920929,0.018252008380373864,0.69997255424705462,0.0,
        0.0,0.0,0.0,0.0,1.0,0.0,-0.0,-0.0,-0.0,-0.0,-0.0,-1.0,-0.0,-0.0,-0.6935356133979842,-0.021630190037277546,
        0.022975637828984145,0.021630190037277546,0.703134798032912,0.0,0.0,0.0,0.0,0.0,1.0,0.0,-0.0,-0.0,-0.0,-0.0,
        -0.0,-1.0,-0.0,-0.0,-0.020191746911356032,-0.69996085369453254,0.026511280680507922,0.69350191818893769,
        0.69996085369453254,0.0,0.0,0.0,0.0,0.0,1.0,0.0,0.0,-0.0,-0.0,-0.0,-0.0,-0.0,-1.0,-0.0,-0.0,
        -0.69999450696241372,-0.022379425814583805,0.023726305453859561,0.609607128237397,0.022379425814583805,0.0,
        0.0,0.0,0.0,0.0,1.0,0.0,0.0,-0.0,-0.0,-0.0,-0.0,-0.0,-1.0,-0.0,0.026511280680507909,-0.6999596977239213,
        0.69350078201899967,0.6999596977239213,0.0,0.0,0.0,0.0,0.0,1.0,0.0,0.0,0.0,-0.0,-0.0,-0.0,-0.0,-0.0,-1.0,
        -0.0,-0.0,0.0223794258145838,0.69996085369453254,-0.02856826556225878,-0.60958947261622121,0.0,0.0,0.0,0.0,
        0.0,1.0,0.0,0.0,0.0,0.0,-0.0,-0.0,-0.0,-0.0,-0.0,-1.0,-0.0,-0.0,0.021630190037277543,-0.69350191818893769,
        -0.027867135223727097,0.703103092376384,0.0,0.0,0.0,0.0,0.0,1.0,0.0,0.0,-0.0,-0.0,-0.0,-0.0,-0.0,-1.0,-0.0,
        -0.0,0.0223794258145838,-0.69996085369453254,-0.02856826556225878,0.60958947261622121,0.0,0.0,0.0,0.0,0.0,
        1.0,0.0,0.0,0.0,-0.0,-0.0,-0.0,-0.0,-0.0,-1.0,-0.0,0.60960712823739716,-0.0224367015618988,
        0.023783898857962432,0.0224367015618988,0.0,0.0,0.0,0.0,0.0,1.0,0.0,0.0,0.0,-0.0,-0.0,-0.0,-0.0,-0.0,-1.0,
        -0.0,0.69997255424705462,-0.023726305453859557,-0.60959621360780769,0.020414853821719429,0.0,0.0,0.0,0.0,
        0.0,1.0,0.0,0.0,-0.0,-0.0,-0.0,-0.0,-0.0,-1.0,-0.0,-0.0,0.69996085369453254,-0.022379425814583808,
        -0.60958947261622132,0.028568265562258718,0.0,0.0,0.0,0.0,0.0,1.0,0.0,0.0,0.0,-0.0,-0.0,-0.0,-0.0,-0.0,-1.0,
        -0.0,-0.0,-0.022975637828984149,-0.69351363803920929,0.019673360677912474,0.703114183187321,0.0,0.0,0.0,0.0,
        0.0,1.0,-0.0,-0.0,-0.0,-0.0,-0.0,-1.0,-0.0,-0.0,-0.026511280680507909,-0.018252008380373868,
        -0.6999596977239213,0.69350078201899967,0.6999596977239213,0.0,0.0,0.0,0.0,0.0,1.0,0.0,0.0,-0.0,-0.0,-0.0,
        -0.0,-0.0,-1.0,-0.0,-0.0,-0.0,-0.023726305453859564,-0.69997255424705462,0.6095962136078078,
        0.020414853821719415,0.0,0.0,0.0,0.0,0.0,1.0,0.0,-0.0,-0.0,-0.0,-0.0,-0.0,-1.0,-0.0,-0.69350191818893769,
        -0.021630190037277546,0.027867135223727094,0.703103092376384,0.0,0.0,0.0,0.0,0.0,1.0,0.0,-0.0,-0.0,-0.0,
        -0.0,-0.0,-1.0,-0.0,-0.0,-0.60960712823739716,-0.703134798032912,-0.0224367015618988,0.023783898857962432,
        0.0224367015618988,0.0,0.0,0.0,0.0,0.0,1.0,0.0,0.0,-0.0,-0.0,-0.0,-0.0,-0.0,-1.0,-0.0,-0.0,-0.0,
        -0.0223794258145838,-0.69996085369453254,0.02856826556225878,0.60958947261622121,0.0,0.0,0.0,0.0,0.0,1.0,
        0.0,0.0,-0.0,-0.0,-0.0,-0.0,-0.0,-1.0,-0.0,0.028568265562258766,0.6999596977239213,-0.609589052036295,0.0,
        0.0,0.0,0.0,0.0,1.0,0.0,0.0,0.0,0.0,-0.0,-0.0,-0.0,-0.0,-0.0,-1.0,-0.0,-0.0,0.027867135223727094,
        -0.69350078201899956,0.02862308593548642,-0.609589052036295,0.0,0.0,0.0,0.0,0.0,1.0,0.0,0.0,0.0,-0.0,-0.0,
        -0.0,-0.0,-0.0,-1.0,-0.0,-0.0,-0.0,0.028568265562258766,-0.6999596977239213,0.609589052036295,0.0,0.0,0.0,
        0.0,0.0,1.0,0.0,0.0,0.0,-0.0,-0.0,-0.0,-0.0,-0.0,-1.0,-0.0,0.60958947261622121,0.022436701561898798,
        -0.028623085935486438,0.0,0.0,0.0,0.0,0.0,1.0,0.0,0.0,0.0,0.0,-0.0,-0.0,-0.0,-0.0,-0.0,-1.0,-0.0,
        0.022436701561898805,-0.60958947261622143,-0.703103092376384,-0.02862308593548641,0.0,0.0,0.0,0.0,0.0,1.0,
        0.0,0.0,0.0,-0.0,-0.0,-0.0,-0.0,-0.0,-1.0,-0.0,-0.0,-0.0,0.6095962136078078,-0.023783898857962432,
        0.609589052036295,-0.028623085935486434,0.0,0.0,0.0,0.0,0.0,1.0,0.0,0.0,0.0,-0.0,-0.0,-0.0,-0.0,-0.0,-1.0,
        -0.0,-0.0,0.60958947261622143,-0.022436701561898795,0.028623085935486438,0.0,0.0,0.0,0.0,0.0,1.0,0.0,0.0,
        0.0,-0.0,-0.0,-0.0,-0.0,-0.0,-1.0,-0.0,0.6999596977239213,-0.028568265562258732,-0.020414853821719432,
        -0.60958905203629477,0.0,0.0,0.0,0.0,0.0,1.0,0.0,0.0,0.0,-0.0,-0.0,-0.0,-0.0,-0.0,-1.0,-0.0,-0.0,-0.0,
        -0.027867135223727094,-0.69350078201899967,-0.019673360677912474,0.70310198599593232,0.0,0.0,0.0,0.0,0.0,
        1.0,0.0,-0.0,-0.0,-0.0,-0.0,-0.0,-1.0,-0.0,-0.0,-0.0,-0.023783898857962435,-0.6095962136078078,
        -0.703114183187321,0.020471261207535715,0.0,0.0,0.0,0.0,0.0,1.0,0.0,-0.0,-0.0,-0.0,-0.0,-0.0,-1.0,-0.0,-0.0,
        -0.0,-0.028568265562258766,-0.020414853821719422,-0.6999596977239213,0.609589052036295,0.0,0.0,0.0,0.0,0.0,
        1.0,0.0,0.0,-0.0,-0.0,-0.0,-0.0,-0.0,-1.0,-0.0,-0.0,-0.60958947261622121,-0.022436701561898798,
        -0.70310309237638391,0.028623085935486438,0.0,0.0,0.0,0.0,0.0,1.0,0.0,0.0,-0.0,-0.0,-0.0,-0.0,-0.0,-1.0,
        -0.0,-0.0,-0.0,0.028623085935486427,0.609589052036295,0.0,0.0,0.0,0.0,0.0,1.0,0.0,0.0,0.0,0.0,-0.0,-0.0,
        -0.0,-0.0,-0.0,-1.0,-0.0,-0.028623085935486427,-0.609589052036295,-0.020471261207535722,
        -0.70310198599593232,0.0,0.0,0.0,0.0,0.0,1.0,0.0,0.0,-0.0,-0.0,-0.0,-0.0,-0.0,-1.0,-0.0,-0.0,-0.0,-0.0,
        0.699842938730663,0.010035599503395155,-0.69332035945645,-0.010841852728168152,-0.699842938730663,
        -0.010035599503395155,0.0,0.0,0.0,0.0,0.0,0.0,0.0,0.0,-0.0,-0.0,-0.0,-0.0,-0.0,-0.0,-0.0,-0.0,
        -0.69984293873066306,0.60877543705459958,0.012215033803492436,-0.012968650442024339,-0.012215033803492436,
        0.0,0.0,0.0,0.0,0.0,0.0,1.0,0.0,0.0,-0.0,-0.0,-0.0,-0.0,-0.0,-0.0,-0.0,-0.0,-0.010035599503395155,
        0.013997402719325952,0.69977736900234788,-0.6932517133063042,-0.69977736900234788,0.0,0.0,0.0,0.0,0.0,0.0,
        0.0,0.0,0.0,-0.0,-0.0,-0.0,-0.0,-0.0,-0.0,-0.0,-0.0,0.6933203594564501,0.01150785335521526,
        -0.0122791159302254,-0.703041617134732,-0.01150785335521526,0.0,0.0,0.0,0.0,0.0,0.0,0.0,-0.0,-0.0,-0.0,-0.0,
        -0.0,-0.0,-0.0,-0.0,0.010841852728168152,0.69980061939953575,-0.69327602991798487,-0.69980061939953575,
        -0.0088862950073843542,0.0,0.0,0.0,0.0,0.0,0.0,0.0,-0.0,-0.0,-0.0,-0.0,-0.0,-0.0,-0.0,-0.0,
        0.69984293873066306,0.012215033803492436,-0.60877543705459958,-0.012968650442024339,-0.012215033803492436,
        0.0,0.0,0.0,0.0,0.0,0.0,0.0,0.0,-0.0,-0.0,-0.0,-0.0,-0.0,-0.0,-1.0,-0.0,0.010035599503395155,
        0.69977736900234788,-0.6932517133063042,-0.013997402719325952,-0.69977736900234788,0.0,0.0,0.0,0.0,0.0,0.0,
        0.0,0.0,-0.0,-0.0,-0.0,-0.0,-0.0,-0.0,-0.0,-0.60877543705459958,0.012283415343526595,-0.0130355444868211,
        -0.012283415343526595,0.0,0.0,0.0,0.0,0.0,0.0,1.0,0.0,0.0,-0.0,-0.0,-0.0,-0.0,-0.0,-0.0,-0.0,-0.0,
        -0.69977736900234788,-0.012215033803492436,0.60871464776796336,0.015705489529037081,0.0,0.0,0.0,0.0,0.0,0.0,
        1.0,0.0,0.0,0.0,-0.0,-0.0,-0.0,-0.0,-0.0,-0.0,-0.0,-0.0,-0.69980061939953575,0.012968650442024337,
        0.60873638906724648,-0.011118767018001796,0.0,0.0,0.0,0.0,0.0,0.0,1.0,0.0,-0.0,-0.0,-0.0,-0.0,-0.0,-0.0,
        -0.0,-0.0,-0.69977736900234788,0.012215033803492436,0.60871464776796336,-0.015705489529037081,0.0,0.0,0.0,
        0.0,0.0,0.0,1.0,0.0,0.0,-0.0,-0.0,-0.0,-0.0,-0.0,-0.0,-0.0,-0.013997402719325936,0.699775564999848,
        -0.69324983267331119,-0.699775564999848,0.0,0.0,0.0,0.0,0.0,0.0,0.0,0.0,0.0,-0.0,-0.0,-0.0,-0.0,-0.0,-0.0,
        -0.0,-0.011507853355215258,0.69325171330630408,0.015154564068334616,-0.70298216286030424,0.0,0.0,0.0,0.0,
        0.0,0.0,0.0,0.0,-0.0,-0.0,-0.0,-0.0,-0.0,-0.0,-0.0,-0.0,-0.012215033803492434,0.69977736900234788,
        0.015705489529037078,-0.60871464776796369,0.0,0.0,0.0,0.0,0.0,0.0,0.0,0.0,0.0,-0.0,-0.0,-0.0,-0.0,-0.0,-0.0,
        -1.0,-0.0,0.69327602991798487,0.0122791159302254,-0.703003309895513,-0.010393624070932634,0.0,0.0,0.0,0.0,
        0.0,0.0,-0.0,-0.0,-0.0,-0.0,-0.0,-0.0,-0.0,-0.0,0.60877543705459958,0.703041617134732,0.012283415343526595,
        -0.0130355444868211,-0.012283415343526595,0.0,0.0,0.0,0.0,0.0,0.0,0.0,0.0,-0.0,-0.0,-0.0,-0.0,-0.0,-0.0,
        -1.0,-0.0,-0.0,0.69325171330630408,0.01150785335521526,-0.015154564068334596,-0.70298216286030424,0.0,0.0,
        0.0,0.0,0.0,0.0,0.0,-0.0,-0.0,-0.0,-0.0,-0.0,-0.0,-0.0,0.012968650442024339,0.69980061939953575,
        -0.60873638906724659,-0.011118767018001793,0.0,0.0,0.0,0.0,0.0,0.0,0.0,-0.0,-0.0,-0.0,-0.0,-0.0,-0.0,-1.0,
        -0.0,0.013997402719325936,0.0088862950073843577,0.699775564999848,-0.69324983267331119,-0.699775564999848,
        0.0,0.0,0.0,0.0,0.0,0.0,0.0,0.0,-0.0,-0.0,-0.0,-0.0,-0.0,-0.0,-0.0,-0.0,-0.0,0.69977736900234788,
        0.012215033803492436,-0.60871464776796336,-0.015705489529037081,0.0,0.0,0.0,0.0,0.0,0.0,0.0,0.0,-0.0,-0.0,
        -0.0,-0.0,-0.0,-0.0,-1.0,-0.60871464776796325,-0.012283415343526595,0.015760046509446644,0.0,0.0,0.0,0.0,
        0.0,0.0,1.0,0.0,0.0,0.0,-0.0,-0.0,-0.0,-0.0,-0.0,-0.0,-0.0,-0.0,-0.60873638906724625,0.013035544486821099,
        -0.60871306985531193,0.015760046509446641,0.0,0.0,0.0,0.0,0.0,0.0,1.0,0.0,0.0,-0.0,-0.0,-0.0,-0.0,-0.0,-0.0,
        -0.0,-0.0,-0.0,-0.60871464776796325,0.012283415343526595,-0.015760046509446644,0.0,0.0,0.0,0.0,0.0,0.0,1.0,
        0.0,0.0,-0.0,-0.0,-0.0,-0.0,-0.0,-0.0,-0.0,-0.015705489529037078,-0.69977556499984794,0.60871306985531193,
        0.0,0.0,0.0,0.0,0.0,0.0,1.0,0.0,0.0,0.0,-0.0,-0.0,-0.0,-0.0,-0.0,-0.0,-0.0,-0.699775564999848,
        0.015705489529037067,0.011118767018001791,0.60871306985531182,0.0,0.0,0.0,0.0,0.0,0.0,1.0,0.0,0.0,-0.0,-0.0,
        -0.0,-0.0,-0.0,-0.0,-0.0,-0.0,-0.0,-0.015154564068334596,0.69324983267331119,-0.015760046509446651,
        0.60871306985531182,0.0,0.0,0.0,0.0,0.0,0.0,0.0,0.0,0.0,-0.0,-0.0,-0.0,-0.0,-0.0,-0.0,-1.0,-0.0,
        -0.015705489529037074,0.699775564999848,-0.60871306985531182,0.0,0.0,0.0,0.0,0.0,0.0,0.0,0.0,0.0,-0.0,-0.0,
        -0.0,-0.0,-0.0,-0.0,-1.0,-0.012283415343526595,0.60871464776796358,0.70298216286030424,0.015760046509446644,
        0.0,0.0,0.0,0.0,0.0,0.0,0.0,0.0,0.0,-0.0,-0.0,-0.0,-0.0,-0.0,-0.0,-1.0,-0.0,-0.0,0.60873638906724625,
        0.013035544486821102,0.703003309895513,-0.011188595264481212,0.0,0.0,0.0,0.0,0.0,0.0,0.0,-0.0,-0.0,-0.0,
        -0.0,-0.0,-0.0,-1.0,-0.0,-0.0,0.69324983267331119,0.015154564068334604,0.010393624070932634,
        -0.70298052278183043,0.0,0.0,0.0,0.0,0.0,0.0,0.0,-0.0,-0.0,-0.0,-0.0,-0.0,-0.0,-0.0,-0.0,-0.0,
        0.60871464776796325,0.70298216286030424,0.012283415343526595,-0.015760046509446644,0.0,0.0,0.0,0.0,0.0,0.0,
        0.0,0.0,-0.0,-0.0,-0.0,-0.0,-0.0,-0.0,-1.0,-0.0,0.015705489529037078,0.69977556499984794,
        0.011118767018001789,-0.60871306985531193,0.0,0.0,0.0,0.0,0.0,0.0,0.0,0.0,-0.0,-0.0,-0.0,-0.0,-0.0,-0.0,
        -1.0,-0.0,-0.0,-0.60871306985531182,-0.015760046509446641,0.0,0.0,0.0,0.0,0.0,0.0,1.0,0.0,0.0,0.0,-0.0,-0.0,
        -0.0,-0.0,-0.0,-0.0,-0.0,0.60871306985531182,0.015760046509446641,0.70298052278183043,0.011188595264481214,
        0.0,0.0,0.0,0.0,0.0,0.0,0.0,0.0,-0.0,-0.0,-0.0,-0.0,-0.0,-0.0,-1.0,-0.0,-0.0,-0.0,0.020191746911356029,
        0.69999450696241372,-0.021532772716851709,-0.6935356133979842,-0.020191746911356029,-0.69999450696241372,
        0.0,0.0,0.0,0.0,0.0,0.0,0.0,0.0,-0.0,-0.0,-0.0,-0.0,-0.0,-0.0,-0.0,-0.0,-0.020191746911356032,
        0.026511280680507922,0.69996085369453254,-0.69350191818893769,-0.69996085369453254,0.0,0.0,0.0,0.0,0.0,0.0,
        0.0,0.0,0.0,-0.0,-0.0,-0.0,-0.0,-0.0,-0.0,-0.0,-0.0,-0.69999450696241372,0.609607128237397,
        0.022379425814583805,-0.023726305453859561,-0.022379425814583805,0.0,0.0,0.0,0.0,0.0,0.0,1.0,0.0,0.0,-0.0,
        -0.0,-0.0,-0.0,-0.0,-0.0,-0.0,-0.0,0.021532772716851712,0.69997255424705462,-0.69351363803920929,
        -0.018252008380373864,-0.69997255424705462,0.0,0.0,0.0,0.0,0.0,0.0,0.0,-0.0,-0.0,-0.0,-0.0,-0.0,-0.0,-0.0,
        -0.0,0.6935356133979842,0.021630190037277546,-0.022975637828984145,-0.021630190037277546,-0.703134798032912,
        0.0,0.0,0.0,0.0,0.0,0.0,0.0,-0.0,-0.0,-0.0,-0.0,-0.0,-0.0,-0.0,-0.0,0.020191746911356032,
        0.69996085369453254,-0.026511280680507922,-0.69350191818893769,-0.69996085369453254,0.0,0.0,0.0,0.0,0.0,0.0,
        0.0,0.0,-0.0,-0.0,-0.0,-0.0,-0.0,-0.0,-0.0,-0.0,0.69999450696241372,0.022379425814583805,
        -0.023726305453859561,-0.609607128237397,-0.022379425814583805,0.0,0.0,0.0,0.0,0.0,0.0,0.0,0.0,-0.0,-0.0,
        -0.0,-0.0,-0.0,-0.0,-0.0,-0.026511280680507909,0.6999596977239213,-0.69350078201899967,-0.6999596977239213,
        0.0,0.0,0.0,0.0,0.0,0.0,0.0,0.0,0.0,-0.0,-0.0,-0.0,-0.0,-0.0,-0.0,-0.0,-0.0,-0.0223794258145838,
        -0.69996085369453254,0.02856826556225878,0.60958947261622121,0.0,0.0,0.0,0.0,0.0,0.0,0.0,1.0,0.0,0.0,-0.0,
        -0.0,-0.0,-0.0,-0.0,-0.0,-0.0,-0.0,-0.021630190037277543,0.69350191818893769,0.027867135223727097,
        -0.703103092376384,0.0,0.0,0.0,0.0,0.0,0.0,0.0,0.0,-0.0,-0.0,-0.0,-0.0,-0.0,-0.0,-0.0,-0.0,
        -0.0223794258145838,0.69996085369453254,0.02856826556225878,-0.60958947261622121,0.0,0.0,0.0,0.0,0.0,0.0,
        0.0,0.0,0.0,-0.0,-0.0,-0.0,-0.0,-0.0,-0.0,-0.0,-0.60960712823739716,0.0224367015618988,
        -0.023783898857962432,-0.0224367015618988,0.0,0.0,0.0,0.0,0.0,0.0,1.0,0.0,0.0,-0.0,-0.0,-0.0,-0.0,-0.0,-0.0,
        -0.0,-0.69997255424705462,0.023726305453859557,0.60959621360780769,-0.020414853821719429,0.0,0.0,0.0,0.0,
        0.0,0.0,1.0,0.0,-0.0,-0.0,-0.0,-0.0,-0.0,-0.0,-0.0,-0.0,-0.69996085369453254,0.022379425814583808,
        0.60958947261622132,-0.028568265562258718,0.0,0.0,0.0,0.0,0.0,0.0,1.0,0.0,0.0,-0.0,-0.0,-0.0,-0.0,-0.0,-0.0,
        -0.0,-0.0,0.022975637828984149,0.69351363803920929,-0.019673360677912474,-0.703114183187321,0.0,0.0,0.0,0.0,
        0.0,0.0,-0.0,-0.0,-0.0,-0.0,-0.0,-0.0,-0.0,-0.0,0.026511280680507909,0.018252008380373868,
        0.6999596977239213,-0.69350078201899967,-0.6999596977239213,0.0,0.0,0.0,0.0,0.0,0.0,0.0,0.0,-0.0,-0.0,-0.0,
        -0.0,-0.0,-0.0,-0.0,-0.0,-0.0,0.023726305453859564,0.69997255424705462,-0.6095962136078078,
        -0.020414853821719415,0.0,0.0,0.0,0.0,0.0,0.0,0.0,-0.0,-0.0,-0.0,-0.0,-0.0,-0.0,-0.0,0.69350191818893769,
        0.021630190037277546,-0.027867135223727094,-0.703103092376384,0.0,0.0,0.0,0.0,0.0,0.0,0.0,-0.0,-0.0,-0.0,
        -0.0,-0.0,-0.0,-0.0,-0.0,0.60960712823739716,0.703134798032912,0.0224367015618988,-0.023783898857962432,
        -0.0224367015618988,0.0,0.0,0.0,0.0,0.0,0.0,0.0,0.0,-0.0,-0.0,-0.0,-0.0,-0.0,-0.0,-1.0,-0.0,-0.0,
        0.0223794258145838,0.69996085369453254,-0.02856826556225878,-0.60958947261622121,0.0,0.0,0.0,0.0,0.0,0.0,
        0.0,0.0,-0.0,-0.0,-0.0,-0.0,-0.0,-0.0,-0.0,-0.028568265562258766,-0.6999596977239213,0.609589052036295,0.0,
        0.0,0.0,0.0,0.0,0.0,0.0,1.0,0.0,0.0,-0.0,-0.0,-0.0,-0.0,-0.0,-0.0,-0.0,-0.0,-0.027867135223727094,
        0.69350078201899956,-0.02862308593548642,0.609589052036295,0.0,0.0,0.0,0.0,0.0,0.0,0.0,0.0,0.0,-0.0,-0.0,
        -0.0,-0.0,-0.0,-0.0,-1.0,-0.0,-0.0,-0.028568265562258766,0.6999596977239213,-0.609589052036295,0.0,0.0,0.0,
        0.0,0.0,0.0,0.0,0.0,0.0,-0.0,-0.0,-0.0,-0.0,-0.0,-0.0,-0.0,-0.60958947261622121,-0.022436701561898798,
        0.028623085935486438,0.0,0.0,0.0,0.0,0.0,0.0,0.0,1.0,0.0,0.0,-0.0,-0.0,-0.0,-0.0,-0.0,-0.0,-0.0,
        -0.022436701561898805,0.60958947261622143,0.703103092376384,0.02862308593548641,0.0,0.0,0.0,0.0,0.0,0.0,0.0,
        0.0,0.0,-0.0,-0.0,-0.0,-0.0,-0.0,-0.0,-1.0,-0.0,-0.0,-0.6095962136078078,0.023783898857962432,
        -0.609589052036295,0.028623085935486434,0.0,0.0,0.0,0.0,0.0,0.0,1.0,0.0,0.0,-0.0,-0.0,-0.0,-0.0,-0.0,-0.0,
        -0.0,-0.0,-0.60958947261622143,0.022436701561898795,-0.028623085935486438,0.0,0.0,0.0,0.0,0.0,0.0,1.0,0.0,
        0.0,-0.0,-0.0,-0.0,-0.0,-0.0,-0.0,-0.0,-0.6999596977239213,0.028568265562258732,0.020414853821719432,
        0.60958905203629477,0.0,0.0,0.0,0.0,0.0,0.0,1.0,0.0,0.0,-0.0,-0.0,-0.0,-0.0,-0.0,-0.0,-0.0,-0.0,-0.0,
        0.027867135223727094,0.69350078201899967,0.019673360677912474,-0.70310198599593232,0.0,0.0,0.0,0.0,0.0,0.0,
        0.0,-0.0,-0.0,-0.0,-0.0,-0.0,-0.0,-0.0,-0.0,-0.0,0.023783898857962435,0.6095962136078078,0.703114183187321,
        -0.020471261207535715,0.0,0.0,0.0,0.0,0.0,0.0,0.0,-0.0,-0.0,-0.0,-0.0,-0.0,-0.0,-1.0,-0.0,-0.0,
        0.028568265562258766,0.020414853821719422,0.6999596977239213,-0.609589052036295,0.0,0.0,0.0,0.0,0.0,0.0,0.0,
        0.0,-0.0,-0.0,-0.0,-0.0,-0.0,-0.0,-0.0,-0.0,0.60958947261622121,0.022436701561898798,0.70310309237638391,
        -0.028623085935486438,0.0,0.0,0.0,0.0,0.0,0.0,0.0,0.0,-0.0,-0.0,-0.0,-0.0,-0.0,-0.0,-0.0,-1.0,-0.0,
        -0.028623085935486427,-0.609589052036295,0.0,0.0,0.0,0.0,0.0,0.0,0.0,1.0,0.0,0.0,-0.0,-0.0,-0.0,-0.0,-0.0,
        -0.0,-0.0,0.028623085935486427,0.609589052036295,0.020471261207535722,0.70310198599593232,0.0,0.0,0.0,0.0,
        0.0,0.0,0.0,0.0,-0.0,-0.0,-0.0,-0.0,-0.0,-0.0,-0.0,-1.0,-0.0,-0.0,0.094300904558948587,
        -0.00035002992429768019,-0.16471311127348245,0.00034173303120953055,-0.094300904558948587,
        0.00035002992429768019,0.0,0.0,0.0,0.0,0.0,0.0,1.0,0.0,-0.0,-0.0,-0.0,-0.0,-0.0,-0.0,-1.0,-0.0,
        -0.0943009045589486,0.49913389863548946,-5.6125427735811955E-5,5.4908765051347066E-5,5.6125427735811955E-5,
        0.0,0.0,0.0,0.0,0.0,0.0,0.0,1.0,0.0,-0.0,-0.0,-0.0,-0.0,-0.0,-0.0,-1.0,-0.0,0.00035002992429768019,
        -0.00027519275766095866,0.09428674239149698,-0.16468822274988468,-0.09428674239149698,0.0,0.0,0.0,0.0,0.0,
        0.0,0.0,1.0,0.0,-0.0,-0.0,-0.0,-0.0,-0.0,-0.0,-1.0,-0.0,0.16471311127348251,4.35775016076801E-20,0.0,0.0,
        -4.35775016076801E-20,0.0,0.0,0.0,0.0,0.0,0.0,0.0,-0.0,-0.0,-0.0,-0.0,-0.0,-0.0,-1.0,-0.0,
        -0.00034173303120953055,0.09429145856464978,-0.16469650149960788,-0.09429145856464978,
        0.00035833304876969549,0.0,0.0,0.0,0.0,0.0,0.0,1.0,-0.0,-0.0,-0.0,-0.0,-0.0,-0.0,-1.0,-0.0,
        0.0943009045589486,-5.6125427735811955E-5,-0.49913389863548946,5.4908765051347066E-5,5.6125427735811955E-5,
        0.0,0.0,0.0,0.0,0.0,0.0,1.0,0.0,-0.0,-0.0,-0.0,-0.0,-0.0,-0.0,-0.0,-0.0,-0.00035002992429768019,
        0.09428674239149698,-0.16468822274988468,0.00027519275766095866,-0.09428674239149698,0.0,0.0,0.0,0.0,0.0,
        0.0,1.0,0.0,-0.0,-0.0,-0.0,-0.0,-0.0,-0.0,-1.0,-0.49913389863548946,4.3575446825768893E-20,0.0,
        -4.3575446825768893E-20,0.0,0.0,0.0,0.0,0.0,0.0,0.0,1.0,0.0,-0.0,-0.0,-0.0,-0.0,-0.0,-0.0,-1.0,-0.0,
        -0.09428674239149698,5.61254277358119E-5,0.49905440057193373,-4.4791776467726323E-5,0.0,0.0,0.0,0.0,0.0,0.0,
        0.0,0.0,1.0,0.0,-0.0,-0.0,-0.0,-0.0,-0.0,-0.0,-1.0,-0.0,-0.09429145856464978,-5.4908765051347025E-5,
        0.49908094429301258,5.7305834211725517E-5,0.0,0.0,0.0,0.0,0.0,0.0,0.0,1.0,-0.0,-0.0,-0.0,-0.0,-0.0,-0.0,
        -1.0,-0.0,-0.09428674239149698,-5.61254277358119E-5,0.49905440057193373,4.4791776467726323E-5,0.0,0.0,0.0,
        0.0,0.0,0.0,0.0,1.0,0.0,-0.0,-0.0,-0.0,-0.0,-0.0,-0.0,-1.0,0.00027519275766095877,0.09428629591571891,
        -0.16468743518794762,-0.09428629591571891,0.0,0.0,0.0,0.0,0.0,0.0,0.0,1.0,0.0,-0.0,-0.0,-0.0,-0.0,-0.0,-0.0,
        -1.0,6.8192497891027074E-21,0.16468822274988465,-4.3243503232001109E-19,-5.188532107227481E-17,0.0,0.0,0.0,
        0.0,0.0,0.0,0.0,0.0,-0.0,-0.0,-0.0,-0.0,-0.0,-0.0,-1.0,-0.0,5.6125427735811887E-5,0.094286742391497008,
        -4.4791776467726296E-5,-0.49905440057193295,0.0,0.0,0.0,0.0,0.0,0.0,0.0,1.0,0.0,-0.0,-0.0,-0.0,-0.0,-0.0,
        -0.0,-0.0,-0.0,0.16469650149960791,0.0,0.0,-1.0114078853662982E-19,0.0,0.0,0.0,0.0,0.0,0.0,-0.0,-0.0,-0.0,
        -0.0,-0.0,-0.0,-1.0,-0.0,0.49913389863548946,0.0,4.3575446825768893E-20,0.0,-4.3575446825768893E-20,0.0,0.0,
        0.0,0.0,0.0,0.0,1.0,0.0,-0.0,-0.0,-0.0,-0.0,-0.0,-0.0,-0.0,-1.0,-0.0,0.16468822274988471,
        4.3577501607680106E-20,0.0,0.0,0.0,0.0,0.0,0.0,0.0,0.0,0.0,-0.0,-0.0,-0.0,-0.0,-0.0,-0.0,-1.0,
        -5.49087650513471E-5,0.0942914585646498,-0.49908094429301236,5.7305834211725388E-5,0.0,0.0,0.0,0.0,0.0,0.0,
        1.0,-0.0,-0.0,-0.0,-0.0,-0.0,-0.0,-0.0,-0.0,-0.00027519275766095877,-0.00035833304876969549,
        0.09428629591571891,-0.16468743518794762,-0.09428629591571891,0.0,0.0,0.0,0.0,0.0,0.0,1.0,0.0,-0.0,-0.0,
        -0.0,-0.0,-0.0,-0.0,-0.0,-1.0,-0.0,0.09428674239149698,-5.61254277358119E-5,-0.49905440057193373,
        4.4791776467726323E-5,0.0,0.0,0.0,0.0,0.0,0.0,1.0,0.0,-0.0,-0.0,-0.0,-0.0,-0.0,-0.0,-0.0,
        -0.49905440057193395,-4.3575446825768893E-20,0.0,0.0,0.0,0.0,0.0,0.0,0.0,0.0,0.0,1.0,0.0,-0.0,-0.0,-0.0,
        -0.0,-0.0,-0.0,-1.0,-0.0,-0.49908094429301275,0.0,-0.49905194196371494,-2.1458936909092391E-19,0.0,0.0,0.0,
        0.0,0.0,0.0,0.0,1.0,0.0,-0.0,-0.0,-0.0,-0.0,-0.0,-0.0,-0.0,-1.0,-0.0,-0.49905440057193395,
        4.3575446825768893E-20,0.0,0.0,0.0,0.0,0.0,0.0,0.0,0.0,1.0,0.0,-0.0,-0.0,-0.0,-0.0,-0.0,-0.0,-1.0,
        4.4791776467726106E-5,-0.09428629591571891,0.49905194196371516,0.0,0.0,0.0,0.0,0.0,0.0,0.0,0.0,1.0,0.0,-0.0,
        -0.0,-0.0,-0.0,-0.0,-0.0,-1.0,-0.09428629591571891,-4.4791776467726174E-5,-5.7305834211725395E-5,
        0.49905194196371527,0.0,0.0,0.0,0.0,0.0,0.0,0.0,1.0,0.0,-0.0,-0.0,-0.0,-0.0,-0.0,-0.0,-0.0,-1.0,-0.0,
        3.71680751054692E-19,0.16468743518794762,3.3854180289225987E-19,0.49905194196371538,0.0,0.0,0.0,0.0,0.0,0.0,
        0.0,1.0,0.0,-0.0,-0.0,-0.0,-0.0,-0.0,-0.0,-0.0,-1.0,4.4791776467726032E-5,0.0942862959157189,
        -0.49905194196371538,0.0,0.0,0.0,0.0,0.0,0.0,0.0,1.0,0.0,-0.0,-0.0,-0.0,-0.0,-0.0,-0.0,-0.0,
        -9.6204993421406312E-20,0.49905440057193323,7.78279816084122E-17,-4.3241746604450817E-19,0.0,0.0,0.0,0.0,
        0.0,0.0,0.0,1.0,0.0,-0.0,-0.0,-0.0,-0.0,-0.0,-0.0,-0.0,-1.0,-0.0,0.49908094429301292,0.0,0.0,
        -1.0113583178806077E-19,0.0,0.0,0.0,0.0,0.0,0.0,1.0,-0.0,-0.0,-0.0,-0.0,-0.0,-0.0,-0.0,-1.0,-0.0,
        0.16468743518794765,-2.1459820267458104E-19,1.0114078853662984E-19,0.0,0.0,0.0,0.0,0.0,0.0,0.0,0.0,-0.0,
        -0.0,-0.0,-0.0,-0.0,-0.0,-0.0,-1.0,-0.0,0.49905440057193395,1.3480376773578907E-22,4.3575446825768893E-20,
        0.0,0.0,0.0,0.0,0.0,0.0,0.0,1.0,0.0,-0.0,-0.0,-0.0,-0.0,-0.0,-0.0,-0.0,-1.0,-4.4791776467726106E-5,
        0.09428629591571891,-5.7305834211725483E-5,-0.49905194196371516,0.0,0.0,0.0,0.0,0.0,0.0,1.0,0.0,-0.0,-0.0,
        -0.0,-0.0,-0.0,-0.0,-0.0,-0.0,-0.0,-0.49905194196371544,2.1458936909092389E-19,0.0,0.0,0.0,0.0,0.0,0.0,0.0,
        0.0,1.0,0.0,-0.0,-0.0,-0.0,-0.0,-0.0,-0.0,-1.0,0.49905194196371544,-2.1458936909092389E-19,
        1.1491477729941819E-22,1.0113583178806082E-19,0.0,0.0,0.0,0.0,0.0,0.0,1.0,0.0,-0.0,-0.0,-0.0,-0.0,-0.0,-0.0,
        -0.0,-0.0,-1.0,-0.0,-0.00034133953126347486,0.09408640843436776,0.0003424380424161977,-0.16434557447790829,
        0.00034133953126347486,-0.09408640843436776,0.0,0.0,0.0,0.0,0.0,0.0,0.0,1.0,-0.0,-0.0,-0.0,-0.0,-0.0,-0.0,
        -0.0,-1.0,0.00034133953126347491,-0.00032196250176989491,0.094072364252867982,-0.16432200077721393,
        -0.094072364252867982,0.0,0.0,0.0,0.0,0.0,0.0,0.0,0.0,1.0,-0.0,-0.0,-0.0,-0.0,-0.0,-0.0,-0.0,-1.0,
        -0.094086408434367746,0.49798249626852653,-4.6869790596096952E-5,4.7137364695702761E-5,
        4.6869790596096952E-5,0.0,0.0,0.0,0.0,0.0,0.0,0.0,0.0,1.0,-0.0,-0.0,-0.0,-0.0,-0.0,-0.0,-0.0,-1.0,
        -0.00034243804241619775,0.094076580236534174,-0.16432907125775337,0.00033721260763744219,
        -0.094076580236534174,0.0,0.0,0.0,0.0,0.0,0.0,1.0,-0.0,-0.0,-0.0,-0.0,-0.0,-0.0,-0.0,-1.0,
        0.16434557447790832,0.0,0.0,0.0,-2.5894641819568537E-17,0.0,0.0,0.0,0.0,0.0,0.0,0.0,-0.0,-0.0,-0.0,-0.0,
        -0.0,-0.0,-0.0,-1.0,-0.00034133953126347491,0.094072364252867982,0.00032196250176989491,
        -0.16432200077721393,-0.094072364252867982,0.0,0.0,0.0,0.0,0.0,0.0,0.0,1.0,-0.0,-0.0,-0.0,-0.0,-0.0,-0.0,
        -0.0,-1.0,0.094086408434367746,-4.6869790596096952E-5,4.7137364695702761E-5,-0.49798249626852653,
        4.6869790596096952E-5,0.0,0.0,0.0,0.0,0.0,0.0,0.0,1.0,-0.0,-0.0,-0.0,-0.0,-0.0,-0.0,-0.0,
        0.00032196250176989475,0.094071772046904353,-0.1643210051126007,-0.094071772046904353,0.0,0.0,0.0,0.0,0.0,
        0.0,0.0,0.0,1.0,-0.0,-0.0,-0.0,-0.0,-0.0,-0.0,-0.0,-1.0,4.68697905960969E-5,-0.094072364252867968,
        -4.4893228007797462E-5,0.49792329220839809,0.0,0.0,0.0,0.0,0.0,0.0,0.0,0.0,0.0,1.0,-0.0,-0.0,-0.0,-0.0,-0.0,
        -0.0,-0.0,-1.0,-6.853661632486371E-20,0.16432200077721393,0.0,2.589093150625205E-17,0.0,0.0,0.0,0.0,0.0,0.0,
        0.0,0.0,-0.0,-0.0,-0.0,-0.0,-0.0,-0.0,-0.0,-1.0,4.68697905960969E-5,0.094072364252867968,
        -4.4893228007797462E-5,-0.49792329220839809,0.0,0.0,0.0,0.0,0.0,0.0,0.0,0.0,1.0,-0.0,-0.0,-0.0,-0.0,-0.0,
        -0.0,-0.0,-0.49798249626852631,0.0,-7.4076964863129346E-20,0.0,0.0,0.0,0.0,0.0,0.0,0.0,0.0,0.0,1.0,-0.0,
        -0.0,-0.0,-0.0,-0.0,-0.0,-0.0,-0.094076580236534188,-4.7137364695702754E-5,0.4979411172906551,
        4.6148095259443704E-5,0.0,0.0,0.0,0.0,0.0,0.0,0.0,1.0,-0.0,-0.0,-0.0,-0.0,-0.0,-0.0,-0.0,-1.0,
        -0.094072364252867968,-4.6869790596096918E-5,0.49792329220839782,4.4893228007797395E-5,0.0,0.0,0.0,0.0,0.0,
        0.0,0.0,0.0,1.0,-0.0,-0.0,-0.0,-0.0,-0.0,-0.0,-0.0,-1.0,2.2880634352910446E-20,0.16432907125775337,
        1.0134306612570304E-19,-2.5892041865377234E-17,0.0,0.0,0.0,0.0,0.0,0.0,-0.0,-0.0,-0.0,-0.0,-0.0,-0.0,-0.0,
        -1.0,-0.00032196250176989475,-0.00033721260763744219,0.094071772046904353,-0.1643210051126007,
        -0.094071772046904353,0.0,0.0,0.0,0.0,0.0,0.0,0.0,1.0,-0.0,-0.0,-0.0,-0.0,-0.0,-0.0,-0.0,-0.0,-1.0,
        -4.7137364695702761E-5,0.094076580236534174,-0.49794111729065493,4.6148095259443779E-5,0.0,0.0,0.0,0.0,0.0,
        0.0,1.0,-0.0,-0.0,-0.0,-0.0,-0.0,-0.0,-0.0,0.16432200077721393,-1.309908514851071E-19,0.0,
        -5.1781863012504081E-17,0.0,0.0,0.0,0.0,0.0,0.0,0.0,-0.0,-0.0,-0.0,-0.0,-0.0,-0.0,-0.0,-1.0,
        0.49798249626852631,7.76839254587056E-17,0.0,-7.4076964863129346E-20,0.0,0.0,0.0,0.0,0.0,0.0,0.0,0.0,1.0,
        -0.0,-0.0,-0.0,-0.0,-0.0,-0.0,-0.0,-0.0,-1.0,-4.68697905960969E-5,0.094072364252867968,
        4.4893228007797462E-5,-0.49792329220839809,0.0,0.0,0.0,0.0,0.0,0.0,0.0,1.0,-0.0,-0.0,-0.0,-0.0,-0.0,-0.0,
        -0.0,4.4893228007797327E-5,-0.094071772046904339,0.49792085025415128,0.0,0.0,0.0,0.0,0.0,0.0,0.0,0.0,0.0,
        1.0,-0.0,-0.0,-0.0,-0.0,-0.0,-0.0,-0.0,-1.0,-2.8648833817456314E-19,0.16432100511260064,
        -4.2251395560396041E-19,0.49792085025415117,0.0,0.0,0.0,0.0,0.0,0.0,0.0,0.0,1.0,-0.0,-0.0,-0.0,-0.0,-0.0,
        -0.0,-0.0,-0.0,-1.0,4.4893228007797327E-5,0.094071772046904339,-0.49792085025415128,0.0,0.0,0.0,0.0,0.0,0.0,
        0.0,0.0,1.0,-0.0,-0.0,-0.0,-0.0,-0.0,-0.0,-0.0,-0.49792329220839782,-4.55642161388578E-20,0.0,0.0,0.0,0.0,
        0.0,0.0,0.0,0.0,0.0,0.0,1.0,-0.0,-0.0,-0.0,-0.0,-0.0,-0.0,-0.0,-8.4301866436910726E-20,0.49792329220839759,
        2.5890931506252044E-17,0.0,0.0,0.0,0.0,0.0,0.0,0.0,0.0,0.0,1.0,-0.0,-0.0,-0.0,-0.0,-0.0,-0.0,-0.0,-0.0,-1.0,
        -0.49794111729065471,1.5354922100091112E-20,-0.49792085025415111,-1.346225068498091E-19,0.0,0.0,0.0,0.0,0.0,
        0.0,0.0,0.0,1.0,-0.0,-0.0,-0.0,-0.0,-0.0,-0.0,-0.0,-0.0,-0.49792329220839765,4.55642161388578E-20,0.0,0.0,
        0.0,0.0,0.0,0.0,0.0,0.0,0.0,1.0,-0.0,-0.0,-0.0,-0.0,-0.0,-0.0,-0.0,-0.094071772046904339,
        -4.4893228007797313E-5,-4.6148095259443785E-5,0.49792085025415139,0.0,0.0,0.0,0.0,0.0,0.0,0.0,0.0,1.0,-0.0,
        -0.0,-0.0,-0.0,-0.0,-0.0,-0.0,-0.0,-1.0,3.4486985836201622E-19,0.16432100511260067,-1.520145991885546E-19,
        -2.5890772937743557E-17,0.0,0.0,0.0,0.0,0.0,0.0,0.0,-0.0,-0.0,-0.0,-0.0,-0.0,-0.0,-0.0,-0.0,-1.0,
        3.681301171504458E-20,0.49794111729065493,-2.589204186537724E-17,2.0267615765916808E-19,0.0,0.0,0.0,0.0,0.0,
        0.0,1.0,-0.0,-0.0,-0.0,-0.0,-0.0,-0.0,-0.0,-0.0,-1.0,-4.4893228007797327E-5,-4.6148095259443833E-5,
        0.094071772046904339,-0.49792085025415128,0.0,0.0,0.0,0.0,0.0,0.0,0.0,1.0,-0.0,-0.0,-0.0,-0.0,-0.0,-0.0,
        -0.0,-0.0,0.49792329220839782,4.55642161388578E-20,7.7672655145631553E-17,0.0,0.0,0.0,0.0,0.0,0.0,0.0,0.0,
        1.0,-0.0,-0.0,-0.0,-0.0,-0.0,-0.0,-0.0,-0.0,-1.0,-5.2483213543760488E-19,-0.49792085025415117,0.0,0.0,0.0,
        0.0,0.0,0.0,0.0,0.0,0.0,1.0,-0.0,-0.0,-0.0,-0.0,-0.0,-0.0,-0.0,5.2483213543760488E-19,0.49792085025415117,
        -1.8142530123302717E-19,-2.5890944949252014E-17,0.0,0.0,0.0,0.0,0.0,0.0,0.0,1.0,-0.0,-0.0,-0.0,-0.0,-0.0,
        -0.0,-0.0,-0.0,-0.0,-1.0];
    Explicit_b_L: ARRAY [0..11] OF LREAL := [0.0001276450955094171,1.2854367351689592E-5,2.3997921309368413E-5,
        8.9335659154009977E-5,0.09512394174964503,1.2151957188376696E-6,2.9283879090142048E-5,
        0.00013338479733282079,9.0052624136951334E-5,2.5990433777560329E-5,-1.5083632311395109E-6,
        0.095123901802077124];
    Explicit_b_Bu: ARRAY [0..11] OF LREAL := [0.013555509581964829,0.00011049700885185901,0.0,0.007544918864475102,
        0.0,0.0,5.9777984595461545E-5,0.013563939607134739,0.0075957283920631228,0.0,0.0,0.0];
    Explicit_b_A: ARRAY [0..35] OF LREAL := [0.99199241976281094,0.0,0.0,0.0,0.0,0.0,0.0,0.9932281507698385,0.0,0.0,
        0.0,0.0,0.015554847722926923,0.0,0.98438237475163026,0.0,0.0,0.0,0.0,0.028694038103379366,0.0,
        0.97120788890393217,0.0,0.0,0.0,0.0,0.0,0.0,1.0,0.0,0.0,0.0,0.0,0.0,0.0,1.0];
    Explicit_b_G: ARRAY [0..67] OF LREAL := [0.0,0.0,10.158815613223508,-0.036771708350285676,-0.036662311053562713,
        9.85465793775906,-1.5299877600979193,0.0031808397609512139,0.0044539458959318295,-2.1419828641370868,
        -0.75929918180634937,0.0027484235492619647,0.003954576204618759,-1.0629716094106481,20.470012239902083,
        -0.043422866829487983,10.152917213237954,9.8495927138850323,10.159519076814444,-2.1419828641370868,
        10.159430876220567,-1.0680198806257994,-0.042190320620619656,19.858017135862909,-1.5299877600979193,
        9.8550853601036952,-0.765177241376307,9.855020081379303,-1.529987760097919,-2.1419828641370873,
        -1.5299877600979193,0.0032455503191138471,-1.5299877600979193,-1.0625325616261672,-0.758582512426614,
        -2.1419828641370868,0.0045508543568839,-2.1419828641370868,-0.758663578393694,-1.0625925131315301,
        20.470012239902079,9.8486646232823229,20.470012239902083,-2.1419828641370873,20.470012239902083,
        -1.0689473852816489,10.152016883575698,19.858017135862916,10.159527486904674,-2.1419828641370868,
        -1.5299877600979195,19.858017135862909,-0.766077082807875,19.858017135862916,-1.529987760097919,
        9.85508888111929,-1.529987760097919,-2.1419828641370877,-1.529987760097919,-2.1419828641370873,
        -1.5299877600979193,-1.0625231274446838,-0.75856647947890077,-2.1419828641370868,20.470012239902079,
        19.858017135862919,-1.5299877600979195,-2.1419828641370873];
    Explicit_b_F: ARRAY [0..679] OF LREAL := [-0.59979259618059289,-0.009353758455642,-0.0906276582768825,
        -0.01119677493626553,-0.59981968570113209,-0.002072221887426051,-9.6629518622770583E-17,
        -0.010600725384405719,-0.59981204597862,0.0,-0.0906276582768825,-0.01119677493626553,-0.59981968570113209,
        -0.002072221887426051,-1.9818538086677218E-16,-0.0112552336137229,-0.090632951151228824,
        -0.0023253378082579569,-0.090631399717964078,9.8255821881498839E-19,-0.090632951151228824,
        -0.0023253378082579569,-0.59982083084269822,2.1684043449710089E-19,-1.6292890498673281E-16,
        -0.0022439033762687364,-0.090632951151228824,-0.0023253378082579556,-1.6912706857826615E-16,
        6.5052130349130266E-19,-1.9818538086677218E-16,-0.0112552336137229,-1.6292424630552291E-16,
        -0.0022439033762687377,-0.090631399717964078,-1.6195269951502222E-18,-0.59982083084269822,
        2.1684043449710089E-19,-0.090632951151228824,-0.0023253378082579569,-1.5277107412502242E-16,
        -0.002333490838741987,-1.9561209477301361E-16,1.7454305018256935E-18,-1.5277107412502242E-16,
        -0.002333490838741987,-0.090633160332066323,1.111307226797642E-18,-0.090633160332066323,
        1.111307226797642E-18,2.1648891582399035E-17,1.6263032587282567E-18,-0.090633160332066323,
        1.111307226797642E-18,-6.6761866353163071E-17,-0.0023334908387419831,-1.1677196210847784E-16,
        3.0182166190834874E-20,-1.466137798731941E-16,-5.4210108624275222E-19,-1.5277107412502242E-16,
        -0.002333490838741987,-0.090633160332066323,1.111307226797642E-18,-8.8415005025334E-17,
        -1.335339788710949E-18,-8.8415005025334E-17,-1.335339788710949E-18,-0.018658322183914295,
        -0.60443870497005736,-0.0039378471707929037,-0.60449198844665231,-0.02056716554843584,-0.091350526032331222,
        -1.3010426069826053E-18,-0.60447749556343533,-0.019915165706996488,1.8932880437028121E-17,
        -0.0039378471707929037,-0.60449198844665231,-0.02056716554843584,-0.091350526032331222,
        -2.6020852139652106E-18,-0.60449452852483609,-0.0042439926459433728,-0.091358640255777612,
        -0.0041398402600447831,1.1931729611497702E-16,-0.0042439926459433728,-0.091358640255777612,
        -0.020617647248818861,2.9287011184264689E-17,-3.7743788129651623E-18,-0.091356412804117382,
        -0.0042439926459433754,-0.0913586402557777,-3.6862873864507151E-18,5.0412012888786939E-17,
        -2.6020852139652106E-18,-0.60449452852483609,-3.4558944247975454E-18,-0.091356412804117465,
        -0.0041398402600447831,-4.7216157578796464E-17,-0.020617647248818861,2.9287011184264689E-17,
        -0.0042439926459433728,-0.091358640255777612,-4.7162794503119443E-18,-0.091359022030849335,
        -3.0357660829594124E-18,2.3489917693256257E-17,-4.7162794503119443E-18,-0.091359022030849335,
        -0.0042522110118177288,6.2083279869003943E-17,-0.0042522110118177288,2.3652886832307984E-16,
        2.0831848895433457E-18,6.1440381862037929E-17,-0.0042522110118177261,6.4481230142680868E-17,
        -7.453889935837843E-20,-0.091359022030849182,-3.2526065174565133E-18,2.3482717913204595E-17,
        -3.0753781081333518E-18,-2.4570731733952744E-17,-4.7162794503119443E-18,-0.091359022030849335,
        -0.0042522110118177288,6.2083279869003943E-17,-2.1752333831413372E-18,9.627400985993671E-18,
        -2.1752333831413372E-18,9.627400985993671E-18,-0.039846405449119417,-0.00070699549145164932,
        -0.0048454234269052479,-0.00083368800678967089,-0.039848507518224073,-0.0001419691362484699,
        -3.5291627747350424E-18,-0.00078983604357177252,-0.039847875544758514,5.4210108624275222E-20,
        -0.0048454234269052479,-0.00083368800678967089,-0.039848507518224073,-0.0001419691362484699,
        -3.0700709173232116E-18,-0.00083681351009234309,-0.0048458257389743867,-0.00015936891402935119,
        -0.0048457020066369596,1.6728900708272432E-19,-0.0048458257389743867,-0.00015936891402935119,
        -0.039848585972544051,2.7105054312137611E-20,-5.6145049513159264E-18,-0.00015337464904168684,
        -0.0048458257389743919,-0.00015936891402935119,-1.5500702934753696E-18,1.4907779871675686E-19,
        -3.0700709173232116E-18,-0.00083681351009234309,-5.6145049513159264E-18,-0.00015337464904168684,
        -0.0048457020066369596,1.2705494208814505E-21,-0.039848585972544051,2.7105054312137611E-20,
        -0.0048458257389743867,-0.00015936891402935119,-2.671475741191059E-18,-0.00015980482794882884,
        -7.1197354381460215E-18,1.1243576553218912E-19,-2.671475741191059E-18,-0.00015980482794882884,
        -0.0048458400753528695,1.0333801956502464E-19,-0.0048458400753528738,2.8629713617195351E-19,
        -2.3776744225020244E-18,-8.1315162936412833E-20,-0.0048458400753528738,1.232432938255007E-19,
        -2.6720977810116989E-18,-0.00015980482794882868,-2.1925447839677564E-18,8.6547907491423286E-20,
        -7.5820301388896576E-18,1.0164395367051604E-19,-2.671475741191059E-18,-0.00015980482794882884,
        -0.0048458400753528695,1.0333801956502464E-19,4.9269050865019288E-18,1.3741949626961802E-19,
        4.9269050865019288E-18,1.3741949626961802E-19,-0.002498588167243714,-0.072033502219620765,
        -0.00048208551817413711,-0.072040801323189754,-0.0027338181113952796,-0.0088047921433480822,
        2.1684043449710089E-19,-0.072038696776594288,-0.0026483714950902354,-4.4740280273972144E-18,
        -0.00048208551817413711,-0.072040801323189754,-0.0027338181113952796,-0.0088047921433480822,
        -2.1684043449710089E-19,-0.07204111228876417,-0.00051981271171570181,-0.0088058927219323933,
        -0.0005061582011700609,-1.4610259548952613E-18,-0.00051981271171570181,-0.0088058927219323933,
        -0.0027386837744431086,5.3600244902252125E-18,-1.1858461261560205E-19,-0.008805574621774134,
        -0.000519812711715702,-0.0088058927219323933,-1.2197274440461925E-19,4.2233062750099415E-18,
        -2.1684043449710089E-19,-0.07204111228876417,-4.4384526436125338E-19,-0.008805574621774134,
        -0.00050615820117006112,-1.1868202140453629E-17,-0.0027386837744431086,5.3600244902252125E-18,
        -0.00051981271171570181,-0.0088058927219323933,-1.3637230450794235E-19,-0.0088059394825071163,
        1.7618285302889447E-19,3.3936375031743543E-18,-1.3637230450794235E-19,-0.0088059394825071163,
        -0.00052060486501435672,2.9797560293222218E-18,-0.00052060486501435607,1.3429019164447288E-17,
        3.3346628342217736E-19,7.9667683854003218E-18,-0.00052060486501435629,3.5800906306887072E-18,
        1.8973538018496328E-19,-0.0088059394825071163,1.2197274440461925E-19,1.3801025446969536E-17,
        -3.34162769497947E-19,-3.085317510373789E-18,-1.3637230450794235E-19,-0.0088059394825071163,
        -0.00052060486501435672,2.9797560293222218E-18,0.0,0.0,0.0,0.0,-4.058413545355279,-0.063594696033629938,
        -0.60907454884520407,-0.076080215252605943,-4.0585979166075674,-0.014036564736267451,6.7713846682582179E-16,
        -0.072032125082489046,-4.0585457813970072,-1.0408340855860843E-17,-0.60907454884520407,
        -0.076080215252605943,-4.0585979166075674,-0.014036564736267451,9.8795212462310378E-16,-0.0764730941294898,
        -0.609110542266128,-0.015751299457167536,-0.60909997131233928,-1.2630955309456127E-17,-0.609110542266128,
        -0.015751299457167536,-4.0586056734283131,-1.0408340855860843E-17,1.0723335468285772E-15,
        -0.015198224064141178,-0.60911054226612926,-0.015751299457167543,1.0873192537314003E-16,
        1.0408340855860843E-17,9.8795212462310378E-16,-0.0764730941294898,4.0616246260380406E-16,
        -0.015198224064141168,-0.60909997131234,-2.076247160309741E-17,-4.0586056734283131,-1.0408340855860843E-17,
        -0.609110542266128,-0.015751299457167536,3.3847436572281842E-16,-0.015806092959488278,
        7.4051008380759953E-17,8.0609213914435577E-18,3.3847436572281842E-16,-0.015806092959488278,
        -0.60911195920864847,-1.1546753136970622E-17,-0.6091119592086478,-3.1983964088322381E-18,
        1.1930103308238973E-15,-7.8062556418956319E-18,-0.6091119592086478,-1.3823577699190182E-17,
        1.7052331768852014E-15,-0.015806092959488267,7.2390823804141524E-16,5.7086314875795605E-18,
        -1.3925391059450148E-16,5.2041704279304213E-18,3.3847436572281842E-16,-0.015806092959488278,
        -0.60911195920864847,-1.1546753136970622E-17,1.3188935306280305E-15,-3.4423618670784138E-18,
        1.3188935306280305E-15,-3.4423618670784138E-18,-0.12604403616769427,-4.0680488499859875,
        -0.026524306561896908,-4.0684090800178625,-0.13890414121671604,-0.61131269070226291,-2.42861286636753E-17,
        -4.0683108951423792,-0.13450295980485635,-5.4784735775692539E-16,-0.026524306561896908,-4.0684090800178625,
        -0.13890414121671604,-0.61131269070226291,-3.6429192995512949E-17,-4.0684261893188367,-0.028586845728186632,
        -0.61136752925546234,-0.027883779531133315,4.99715557562147E-16,-0.028586845728186632,-0.61136752925546234,
        -0.13924196197629707,5.7842185902101662E-17,-4.6187012547882489E-17,-0.61135244809992562,
        -0.028586845728186632,-0.61136752925546234,-2.7755575615628914E-17,7.1077583922718457E-16,
        -3.6429192995512949E-17,-4.0684261893188367,-2.5370330836160804E-17,-0.61135244809992562,
        -0.027883779531133336,-8.463553208964969E-16,-0.13924196197629707,5.7842185902101662E-17,
        -0.028586845728186632,-0.61136752925546234,-5.0523821237824507E-17,-0.61137010083038879,
        -2.8622937353617317E-17,6.4463442450788527E-16,-5.0523821237824507E-17,-0.61137010083038879,
        -0.028641842628589886,-2.7770822208679491E-16,-0.028641842628589844,4.1030275964998308E-16,
        -5.6753325048406258E-18,-1.2061749168901237E-16,-0.028641842628589886,-2.5845685726159917E-16,
        -5.3668007538032469E-17,-0.61137010083038823,-2.7755575615628914E-17,-3.5405977195229754E-17,
        -2.6492014216562311E-17,-1.2059038663470023E-16,-5.0523821237824507E-17,-0.61137010083038879,
        -0.028641842628589886,-2.7770822208679491E-16,-4.7145143278842451E-19,1.9176338982052209E-17,
        -4.7145143278842451E-19,1.9176338982052209E-17,4.058413545355279,0.063594696033629938,0.60907454884520407,
        0.076080215252605943,4.0585979166075674,0.014036564736267451,-6.7713846682582179E-16,0.072032125082489046,
        4.0585457813970072,1.0408340855860843E-17,0.60907454884520407,0.076080215252605943,4.0585979166075674,
        0.014036564736267451,-9.8795212462310378E-16,0.0764730941294898,0.609110542266128,0.015751299457167536,
        0.60909997131233928,1.2630955309456127E-17,0.609110542266128,0.015751299457167536,4.0586056734283131,
        1.0408340855860843E-17,-1.0723335468285772E-15,0.015198224064141178,0.60911054226612926,
        0.015751299457167543,-1.0873192537314003E-16,-1.0408340855860843E-17,-9.8795212462310378E-16,
        0.0764730941294898,-4.0616246260380406E-16,0.015198224064141168,0.60909997131234,2.076247160309741E-17,
        4.0586056734283131,1.0408340855860843E-17,0.609110542266128,0.015751299457167536,-3.3847436572281842E-16,
        0.015806092959488278,-7.4051008380759953E-17,-8.0609213914435577E-18,-3.3847436572281842E-16,
        0.015806092959488278,0.60911195920864847,1.1546753136970622E-17,0.6091119592086478,3.1983964088322381E-18,
        -1.1930103308238973E-15,7.8062556418956319E-18,0.6091119592086478,1.3823577699190182E-17,
        -1.7052331768852014E-15,0.015806092959488267,-7.2390823804141524E-16,-5.7086314875795605E-18,
        1.3925391059450148E-16,-5.2041704279304213E-18,-3.3847436572281842E-16,0.015806092959488278,
        0.60911195920864847,1.1546753136970622E-17,-1.3188935306280305E-15,3.4423618670784138E-18,
        -1.3188935306280305E-15,3.4423618670784138E-18,0.12604403616769427,4.0680488499859875,0.026524306561896908,
        4.0684090800178625,0.13890414121671604,0.61131269070226291,2.42861286636753E-17,4.0683108951423792,
        0.13450295980485635,5.4784735775692539E-16,0.026524306561896908,4.0684090800178625,0.13890414121671604,
        0.61131269070226291,3.6429192995512949E-17,4.0684261893188367,0.028586845728186632,0.61136752925546234,
        0.027883779531133315,-4.99715557562147E-16,0.028586845728186632,0.61136752925546234,0.13924196197629707,
        -5.7842185902101662E-17,4.6187012547882489E-17,0.61135244809992562,0.028586845728186632,0.61136752925546234,
        2.7755575615628914E-17,-7.1077583922718457E-16,3.6429192995512949E-17,4.0684261893188367,
        2.5370330836160804E-17,0.61135244809992562,0.027883779531133336,8.463553208964969E-16,0.13924196197629707,
        -5.7842185902101662E-17,0.028586845728186632,0.61136752925546234,5.0523821237824507E-17,0.61137010083038879,
        2.8622937353617317E-17,-6.4463442450788527E-16,5.0523821237824507E-17,0.61137010083038879,
        0.028641842628589886,2.7770822208679491E-16,0.028641842628589844,-4.1030275964998308E-16,
        5.6753325048406258E-18,1.2061749168901237E-16,0.028641842628589886,2.5845685726159917E-16,
        5.3668007538032469E-17,0.61137010083038823,2.7755575615628914E-17,3.5405977195229754E-17,
        2.6492014216562311E-17,1.2059038663470023E-16,5.0523821237824507E-17,0.61137010083038879,
        0.028641842628589886,2.7770822208679491E-16,4.7145143278842451E-19,-1.9176338982052209E-17,
        4.7145143278842451E-19,-1.9176338982052209E-17,-0.035836878619887123,-0.0020044921093567546,
        -0.500620860139117,-0.00032212069274566483,-0.035843309272630818,-0.00027596269360220414,-1.0,0.0,
        -0.035841046673494539,-1.8973538018496328E-19,-0.500620860139117,-0.00032212069274566483,
        -0.035843309272630818,-0.00027596269360220414,-1.0,0.0,-0.50062102552106991,-4.4922425567013027E-5,
        -0.500620967776861,-6.5052130349130266E-19,-0.50062102552106991,-4.4922425567013027E-5,
        -0.035843461773843677,1.2197274440461925E-19,-0.99999999999999978,-4.3368086899420177E-19,
        -0.50062102552106991,-4.4922425567013027E-5,-1.0,0.0,-1.0,0.0,-1.0,0.0,-0.500620967776861,0.0,
        -0.035843461773843677,1.2197274440461925E-19,-0.50062102552106991,-4.4922425567013027E-5,-1.0,0.0,-1.0,0.0,
        -1.0,0.0,-0.5006210295621647,-4.3368086899420177E-19,-0.50062102956216481,-2.1684043449710089E-19,
        -1.0000000000000002,0.0,-0.5006210295621647,-4.3368086899420177E-19,-0.99999999999999978,0.0,-1.0,0.0,-1.0,
        0.0,-1.0,0.0,-0.5006210295621647,-4.3368086899420177E-19,-1.0,0.0,-1.0,0.0,-0.0020044921093567546,
        -0.03600361345613274,-0.00032212069274566456,-0.036009703110027817,-0.00027596269360220414,
        -0.500624245328719,-2.7105054312137611E-19,-0.036007780788949534,0.0,-1.0,-0.00032212069274566456,
        -0.036009703110027817,-0.00027596269360220414,-0.500624245328719,-3.2526065174565133E-19,
        -0.036009910891515694,-4.492242556701281E-5,-0.500624360178471,0.0,-1.0000000000000002,
        -4.492242556701281E-5,-0.500624360178471,0.0,-0.99999999999999978,0.0,-0.50062432431526649,
        -4.4922425567012376E-5,-0.500624360178471,0.0,-1.0,-3.2526065174565133E-19,-0.036009910891515694,
        -2.1684043449710089E-19,-0.50062432431526638,4.3368086899420177E-19,-0.99999999999999978,0.0,
        -0.99999999999999978,-4.492242556701281E-5,-0.500624360178471,-2.1684043449710089E-19,-0.50062436421953882,
        0.0,-1.0,-2.1684043449710089E-19,-0.50062436421953882,-4.3368086899420177E-19,-0.99999999999999978,0.0,
        -1.0000000000000002,0.0,-0.99999999999999978,-4.3368086899420177E-19,-0.99999999999999978,
        -2.1684043449710089E-19,-0.50062436421953893,0.0,-1.0,-8.6736173798840355E-19,-1.0,-2.1684043449710089E-19,
        -0.50062436421953882,-4.3368086899420177E-19,-0.99999999999999978,-8.6736173798840355E-19,-1.0,
        -8.6736173798840355E-19,-1.0];
END_VAR

VAR_TEMP
    new_x: ARRAY [0..5] OF LREAL;
    y_innov: ARRAY [0..1] OF LREAL;
    th: ARRAY [0..9] OF LREAL;
    b_k: DINT;
    du: ARRAY [0..1] OF LREAL;
    found: BOOL;
    regionmin: DINT;
    betamin: LREAL;
    beta: LREAL;
    betah: LREAL;
    b_h: DINT;
    rtb_xest: ARRAY [0..5] OF LREAL;
    i: DINT;
    rtb_last_mv_idx_0: LREAL;
    rtb_last_mv_idx_1: LREAL;
END_VAR

CASE ssMethodType OF
    SS_INITIALIZE: 
        (* SystemInitialize for Atomic SubSystem: '<Root>/Explicit Controller' *)
        (* InitializeConditions for Memory: '<S3>/last_x' *)
        FOR i := 0 TO 5 DO 
            last_x_PreviousInput[i] := 0.0;
        END_FOR;
        (* End of InitializeConditions for Memory: '<S3>/last_x' *)
        
        (* InitializeConditions for UnitDelay: '<S3>/last_mv' *)
        last_mv_DSTATE[0] := 0.0;
        last_mv_DSTATE[1] := 0.0;
        (* End of SystemInitialize for SubSystem: '<Root>/Explicit Controller' *)
    SS_STEP: 
        rtb_last_mv_idx_0 := last_mv_DSTATE[0];
        rtb_last_mv_idx_1 := last_mv_DSTATE[1];
        regionmin := 1;
        b_k := -1;
        (* End of Outputs for SubSystem: '<Root>/Explicit Controller' *)
        (* Outputs for Atomic SubSystem: '<Root>/Explicit Controller' *)
        (* MATLAB Function: '<S3>/Explicit MPC Evaluation' incorporates:
         *  Memory: '<S3>/last_x' *)
        FOR i := 0 TO 5 DO 
            new_x[i] := last_x_PreviousInput[i];
        END_FOR;
        (* End of Outputs for SubSystem: '<Root>/Explicit Controller' *)
        (* Outputs for Atomic SubSystem: '<Root>/Explicit Controller' *)
        (* MATLAB Function: '<S3>/Explicit MPC Evaluation' *)
        FOR i := 0 TO 1 DO 
            betamin := 0.0;
            FOR b_h := 0 TO 5 DO 
                betamin := (Explicit_b_Cm[(b_h * 2) + i] * new_x[b_h]) + betamin;
            END_FOR;
            y_innov[i] := MeasuredTankOutputs[i] - betamin;
        END_FOR;
        (* End of Outputs for SubSystem: '<Root>/Explicit Controller' *)
        (* Outputs for Atomic SubSystem: '<Root>/Explicit Controller' *)
        (* MATLAB Function: '<S3>/Explicit MPC Evaluation' *)
        FOR i := 0 TO 5 DO 
            rtb_xest[i] := ((Explicit_b_M[i + 6] * y_innov[1]) + (Explicit_b_M[i] * y_innov[0])) + new_x[i];
        END_FOR;
        (* End of Outputs for SubSystem: '<Root>/Explicit Controller' *)
        (* Outputs for Atomic SubSystem: '<Root>/Explicit Controller' *)
        (* MATLAB Function: '<S3>/Explicit MPC Evaluation' *)
        FOR i := 0 TO 9 DO 
            th[i] := 0.0;
        END_FOR;
        FOR b_h := 0 TO 5 DO 
            th[b_h] := rtb_xest[b_h];
        END_FOR;
        th[6] := ref[0];
        th[8] := rtb_last_mv_idx_0;
        th[7] := ref[1];
        th[9] := rtb_last_mv_idx_1;
        FOR b_h := 0 TO 9 DO 
            betamin := th[b_h];
            IF betamin < Explicit_b_thmin[b_h] THEN 
                regionmin := 0;
            ELSIF betamin > Explicit_b_thmax[b_h] THEN 
                regionmin := 0;
            END_IF;
        END_FOR;
        du[0] := 0.0;
        du[1] := 0.0;
        IF regionmin = 1 THEN 
            found := FALSE;
            regionmin := 0;
            betamin := 1.797693134862316E+307;
            WHILE ( NOT found) AND ((b_k + 1) < 34) DO
                b_k := b_k + 1;
                b_h := INT_TO_DINT(b_i1[b_k]);
                beta := -1.0;
                WHILE b_h <= INT_TO_DINT(b_i2[b_k]) DO
                    betah := 0.0;
                    FOR i := 0 TO 9 DO 
                        betah := (Explicit_g_H[((697 * i) + b_h) - 1] * th[i]) + betah;
                    END_FOR;
                    betah := betah - Explicit_c_K[b_h - 1];
                    IF betah > beta THEN 
                        beta := betah;
                    END_IF;
                    b_h := b_h + 1;
                END_WHILE;
                IF beta <= 0.0 THEN 
                    found := TRUE;
                ELSIF betamin > beta THEN 
                    betamin := beta;
                    regionmin := b_k + 1;
                END_IF;
            END_WHILE;
            IF  NOT found THEN 
                b_k := regionmin - 1;
            END_IF;
            b_k := DWORD_TO_DINT(SHL(DINT_TO_DWORD(b_k), 1));
            FOR regionmin := 0 TO 1 DO 
                b_h := regionmin + b_k;
                betamin := 0.0;
                FOR i := 0 TO 9 DO 
                    betamin := (Explicit_b_F[(68 * i) + b_h] * th[i]) + betamin;
                END_FOR;
                du[regionmin] := Explicit_b_G[regionmin + b_k] + betamin;
            END_FOR;
        END_IF;
        rtb_last_mv_idx_0 := rtb_last_mv_idx_0 + du[0];
        betamin := rtb_last_mv_idx_0;
        mv[0] := rtb_last_mv_idx_0;
        rtb_last_mv_idx_0 := rtb_last_mv_idx_1 + du[1];
        mv[1] := rtb_last_mv_idx_0;
        (* End of Outputs for SubSystem: '<Root>/Explicit Controller' *)
        (* Outputs for Atomic SubSystem: '<Root>/Explicit Controller' *)
        FOR i := 0 TO 5 DO 
            (* MATLAB Function: '<S3>/Explicit MPC Evaluation' *)
            rtb_xest[i] := 0.0;
            FOR b_h := 0 TO 5 DO 
                rtb_xest[i] := (Explicit_b_A[(6 * b_h) + i] * new_x[b_h]) + rtb_xest[i];
            END_FOR;
            (* Update for Memory: '<S3>/last_x' incorporates:
             *  MATLAB Function: '<S3>/Explicit MPC Evaluation' *)
            last_x_PreviousInput[i] := ((Explicit_b_L[i + 6] * y_innov[1]) + (Explicit_b_L[i] * y_innov[0])) + (rtb_xest[i] + ((Explicit_b_Bu[i + 6] * rtb_last_mv_idx_0) + (Explicit_b_Bu[i] * betamin)));
        END_FOR;
        (* Update for UnitDelay: '<S3>/last_mv' *)
        last_mv_DSTATE[0] := mv[0];
        last_mv_DSTATE[1] := rtb_last_mv_idx_0;
        (* End of Outputs for SubSystem: '<Root>/Explicit Controller' *)
END_CASE;

END_FUNCTION_BLOCK

(* stored: Version 1.1.0.1, ProductVersion 3.1.4024.5
   POU Explicit_Controller_FCN_BLK: Id {5ccb6c6a-4b07-466d-8aa3-23f01e644d56}, SpecialFunc None *)
